		07: GEO.IP4 := IP4_DECODE(STR:=CTRL.VALUE); (* IP-Adresse *)
		10: GEO.STATE := 'OK' = CTRL.VALUE; (* STATUS *)
		13: GEO.COUNTRY_CODE := CTRL.VALUE; (* Country-Code *)
		16: GEO.COUNTRY_NAME := CTRL.VALUE; (* Country-Name *)
		19: GEO.REGION_CODE := CTRL.VALUE; (* Region-Code *)
		22: GEO.REGION_NAME := CTRL.VALUE; (* Region-Name *)
		25: GEO.CITY := CTRL.VALUE; (* City *)
		31: GEO.GEO_LATITUDE := value_real; (* Latitude *)
		34: GEO.GEO_LONGITUDE := value_real; (* Longitude *)
		37: GEO.TIME_ZONE_NAME := CTRL.VALUE; (* TimeZone Name *)
		40: GEO.GMT_OFFSET := value_int; (* GMT OFFSET in Sekunden *)
		43: GEO.IS_DST := value_int > 0; (* Sommerzeit aktiv *)
		END_CASE;

	ELSIF CTRL.TYP = 99 THEN (* EXIT - letztes Element gelesen *)
		DONE := TRUE;
		state := 100;
	END_IF;

100:
	(* UNLOCK HTTP DATA *)
	IF (NOT HTTP_GET.DONE) THEN
		state := 0;
		BUSY := FALSE;
		DONE := ERROR_T = BYTE#0;
	END_IF;

END_CASE;

(* ---------------- DNS --------------- *)
DNS_CLIENT(	IP_C:=IP_C,
			S_BUF:=S_BUF,
			R_BUF:=R_BUF,
			DOMAIN:=URL_DATA.DOMAIN,
			IP4_DNS:=DWORD#00,
			ACTIVATE:=state=40 (* DNS Start *)
			);

(* nicht oder nicht direkt verwendete Parameter *)
(* 	DWORD :=DNS_CLIENT.IP4;
	BOOL  :=DNS_CLIENT.DONE;
	BYTE  :=DNS_CLIENT.ERROR; *)
(* -------------------------------------*)

(* ------------- HTTP_GET --------------- *)
HTTP_GET(	IP_C:=IP_C,
			S_BUF:=S_BUF,
			R_BUF:=R_BUF,
			IP4:=DNS_CLIENT.IP4,
			GET:=state=60,
			MODE:=BYTE#2, (* HTTP 1.1 mit persistenter Verbindung *)
			UNLOCK_BUF:=state=100,
			URL_DATA:=URL_DATA
			);

(* nicht oder nicht direkt verwendete Parameter *)
(*	STRING := HTTP_GET.HTTP_STATUS;
	UINT :=HTTP_GET.HEADER_START;
	UINT :=HTTP_GET.HEADER_STOP;
	UINT :=HTTP_GET.BODY_START;
	UINT :=HTTP_GET.BODY_STOP;
	BOOL :=HTTP_GET.DONE;
	BYTE :=HTTP_GET.ERROR;
*)
(* -------------------------------------*)

last_state := ACTIVATE;

(* revision history
ks	14. aug. 2009	rev 1.0
	original version

ks	07. oct. 2010	rev 1.1
	new url , ip2geo fields , REAL_CHECK
*)

END_FUNCTION_BLOCK

// POUs/DEMO/IP2GEO_DEMO
PROGRAM IP2GEO_DEMO
VAR
	IP_C: IP_C;
	S_BUF: NETWORK_BUFFER;
	R_BUF: NETWORK_BUFFER;
	IP_CONTROL_1: IP_CONTROL;
	CLK_PRG : oscat_basic.CLK_PRG;
	IP2GEO_1: IP2GEO;
	GEO: IP2GEO_DATA;
	activate: BOOL := TRUE;
	done: BOOL;
	busy: BOOL;
	error_c: DWORD;
	error_t: BYTE;
END_VAR
VAR // added by the converter: edge detectors and wires of the graphical bodies
    _w1 : ANY;
END_VAR

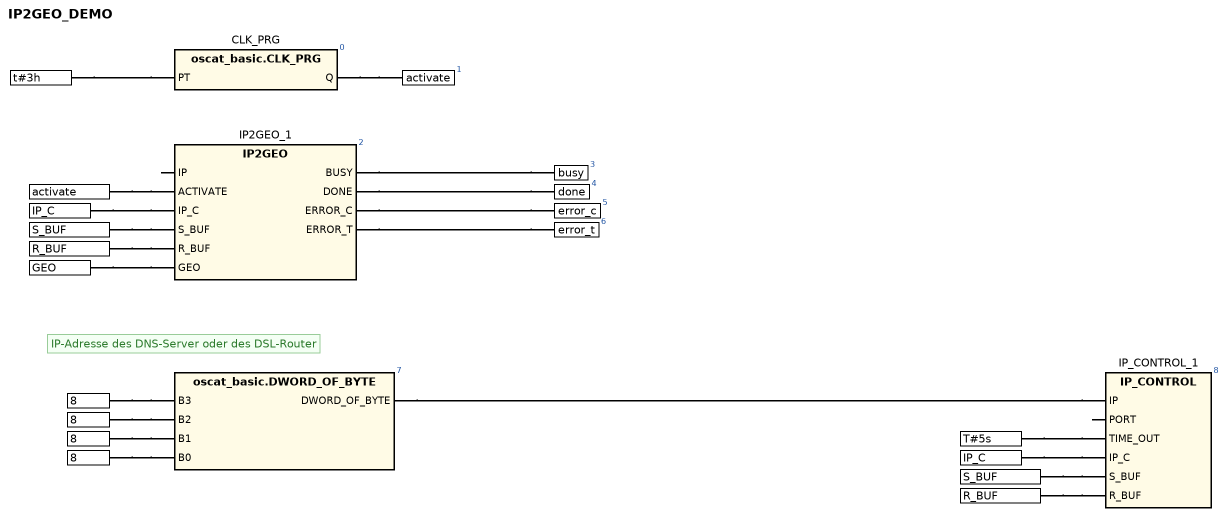
CLK_PRG(PT := t#3h); // oscat_basic.CLK_PRG
activate := CLK_PRG.Q;
IP2GEO_1(ACTIVATE := activate, IP_C := IP_C, S_BUF := S_BUF, R_BUF := R_BUF, GEO := GEO); // IP2GEO
busy := IP2GEO_1.BUSY;
done := IP2GEO_1.DONE;
error_c := IP2GEO_1.ERROR_C;
error_t := IP2GEO_1.ERROR_T;
// IP-Adresse des DNS-Server oder des DSL-Router
_w1 := oscat_basic.DWORD_OF_BYTE(B3 := 8, B2 := 8, B1 := 8, B0 := 8);
IP_CONTROL_1(IP := _w1, TIME_OUT := T#5s, IP_C := IP_C, S_BUF := S_BUF, R_BUF := R_BUF); // IP_CONTROL

END_PROGRAM

// POUs/CONVERT/IP4_CHECK
FUNCTION IP4_CHECK : BOOL
VAR_INPUT
	NIP : DWORD;
	LIP : DWORD;
	SM : DWORD;
END_VAR


(*
version 1.0	4. mar 2008
programmer 	hugo
tested by		oscat

IP4_CHECK testet ob eine Network IP und Local_IP im selben Subnet sind.

*)

IP4_CHECK := (NIP AND sm) = (LIP AND SM);


(* revision history
hm		4. mar 2008	rev 1.0
	original version

*)

END_FUNCTION

// POUs/DRIVER/IRTRANS_DECODE
FUNCTION_BLOCK IRTRANS_DECODE
VAR_IN_OUT
	IP_C : IP_C; (* IP_Control Verwaltungsstruktur *)
	R_BUF : NETWORK_BUFFER_SHORT;
END_VAR
VAR_OUTPUT
	CMD : BOOL;
	DEV : STRING;
	KEY : STRING;
	ERROR : BOOL;
END_VAR
VAR
	i : INT;
	stop : INT;
	pt : POINTER TO BYTE;
	buffer : POINTER TO ARRAY[0..32000] OF BYTE;
	size : UINT;
	z : BYTE;
END_VAR

(*

version 1.2		06. dec. 2009
programmer 		ks
tested by		ks

*)

size := R_BUF.SIZE;

(* do nothing if the buffer is empty *)
IF size > 0 AND IP_C.MAILBOX[1] <> z THEN
	i := 0;
	error := TRUE;
	stop := size - 2;
	(* read characters before first comma and store in device *)
	pt := ADR(dev);
	buffer := ADR(R_BUF.BUFFER);
	WHILE i < stop DO
		IF buffer^[i] = 44 THEN EXIT; END_IF;
		pt^ := buffer^[i];
		pt := pt + 1;
		i := i + 1;
	END_WHILE;
	(* terminate the device string *)
	pt^ := 0;
	(* read after first comma and store in key *)
	i := i + 1;
	pt := ADR(key);
	WHILE i < stop DO
		pt^ := buffer^[i];
		pt := pt + 1;
		i := i + 1;
	END_WHILE;
	(* terminate the key string *)
	pt^:= 0;
	(* check if last two characters are $R$N 13, 10 *)
	IF buffer^[i] <> 13 AND buffer^[i+1] <> 10 THEN	RETURN;	END_IF;
	(* check if device and key are present *)
	IF LEN(dev) = 0 OR LEN(key) = 0 THEN RETURN; END_IF;
	(* a valid transmission has been received *)
	cmd := TRUE;
	error := FALSE;
ELSE
	error := FALSE;
	cmd := FALSE;
END_IF;

z := IP_C.MAILBOX[1];

(* revision history
ks	18. oct. 2008	rev 1.0
	original version
ks	20. oct. 2009	rev 1.1
	Networkbuffer und Buffer-funktionen auf Basis 0
ks	06. dec. 2009	rev 1.2
	Codeanpassung für IRTRANS_SERVER
*)

END_FUNCTION_BLOCK

// POUs/DRIVER/IRTRANS_SERVER
FUNCTION_BLOCK IRTRANS_SERVER
VAR_IN_OUT
	IP_C : IP_C; (* IP_Control Verwaltungsstruktur *)
	S_BUF : NETWORK_BUFFER_SHORT;
	R_BUF : NETWORK_BUFFER_SHORT;
END_VAR
VAR_INPUT
	UDP_TCP : BOOL;
END_VAR
VAR_OUTPUT
	S_ENABLE : BOOL;
	R_ENABLE : BOOL;
	ERROR : DWORD;
END_VAR
VAR
	t : TON;
END_VAR

(*
version 1.1		17. may. 2011
programmer 		ks
tested by			ks
*)

IF NOT IP_C.C_ENABLE THEN
	(* IP Datenverkehr einrichten *)
	IP_C.C_PORT := WORD#0; (* Portnummer eintragen *)
	IP_C.C_IP := DWORD#00; (* IP eintragen *)
	IP_C.C_MODE := SEL(UDP_TCP,5,4); (* 4 = Mode: TCP+PASSIV+PORT / 5 = Mode: UDP+PASSIV+PORT*)
	IP_C.C_ENABLE := TRUE; (* Verbindungsaufbau freigeben *)
	IP_C.R_OBSERVE := FALSE; (* Datenempfang ueberwachen *)
	IP_C.TIME_RESET := TRUE; (* Zeitueberwachung rücksetzen *)
	S_BUF.SIZE := UINT#0; (* Sendedaten rücksetzen *)
	R_BUF.SIZE := UINT#0; (* Empfangsdaten rücksetzen *)
END_IF;

R_ENABLE := IP_C.C_STATE > 127;
S_ENABLE := R_ENABLE AND (IP_C.MAILBOX[1] > 0 OR IP_C.C_MODE <> 5);
ERROR := IP_C.ERROR;

t(IN:= IP_C.ERROR > 0, PT:=T#5s);
IF t.Q THEN
	IP_C.TIME_RESET := TRUE; (* Error Reset *)
END_IF;

(* revision history
ks	6. dec 2009		rev 1.0
	original version

ks	17. may 2011		rev 1.1
	neue Fehlerausgabe und Empfangsbuffer rücksetzen
*)

END_FUNCTION_BLOCK

// POUs/DEMO/IRTRANS_DEMO
PROGRAM IRTRANS_DEMO
VAR
	IP_C : IP_C;
	S_BUF : NETWORK_BUFFER_SHORT;
	R_BUF : NETWORK_BUFFER_SHORT;
	IP_CONTROL2 : IP_CONTROL2;
	IRTRANS_DECODE : IRTRANS_DECODE;
	IRTRANS_RCV_4 : IRTRANS_RCV_4;
	DRIVER_4 : oscat_basic.DRIVER_4;
	IRTRANS_SERVER : IRTRANS_SERVER;
	IRTRANS_SND_8_1 : IRTRANS_SND_8;
	IRTRANS_SND_8_2 : IRTRANS_SND_8;
	Q0: BOOL;
	Q1: BOOL;
	Q2: BOOL;
	Q3: BOOL;
	error: BOOL;
	error_server: DWORD;
	Send_1_0: BOOL := TRUE;
	Send_1_1: BOOL;
	Send_1_2: BOOL;
	Send_1_3: BOOL;
	Send_1_4: BOOL;
	Send_1_5: BOOL;
	Send_1_6: BOOL;
	Send_1_7: BOOL;
	Send_2_0: BOOL := TRUE;
	Send_2_1: BOOL;
	Send_2_2: BOOL;
	Send_2_3: BOOL;
	Send_2_4: BOOL;
	Send_2_5: BOOL;
	Send_2_6: BOOL;
	Send_2_7: BOOL;
	R_ENABLE: BOOL;
	S_ENABLE: BOOL;
	MODE: BOOL := FALSE;
	KEY_1: BYTE;
	KEY_2: BYTE;
END_VAR

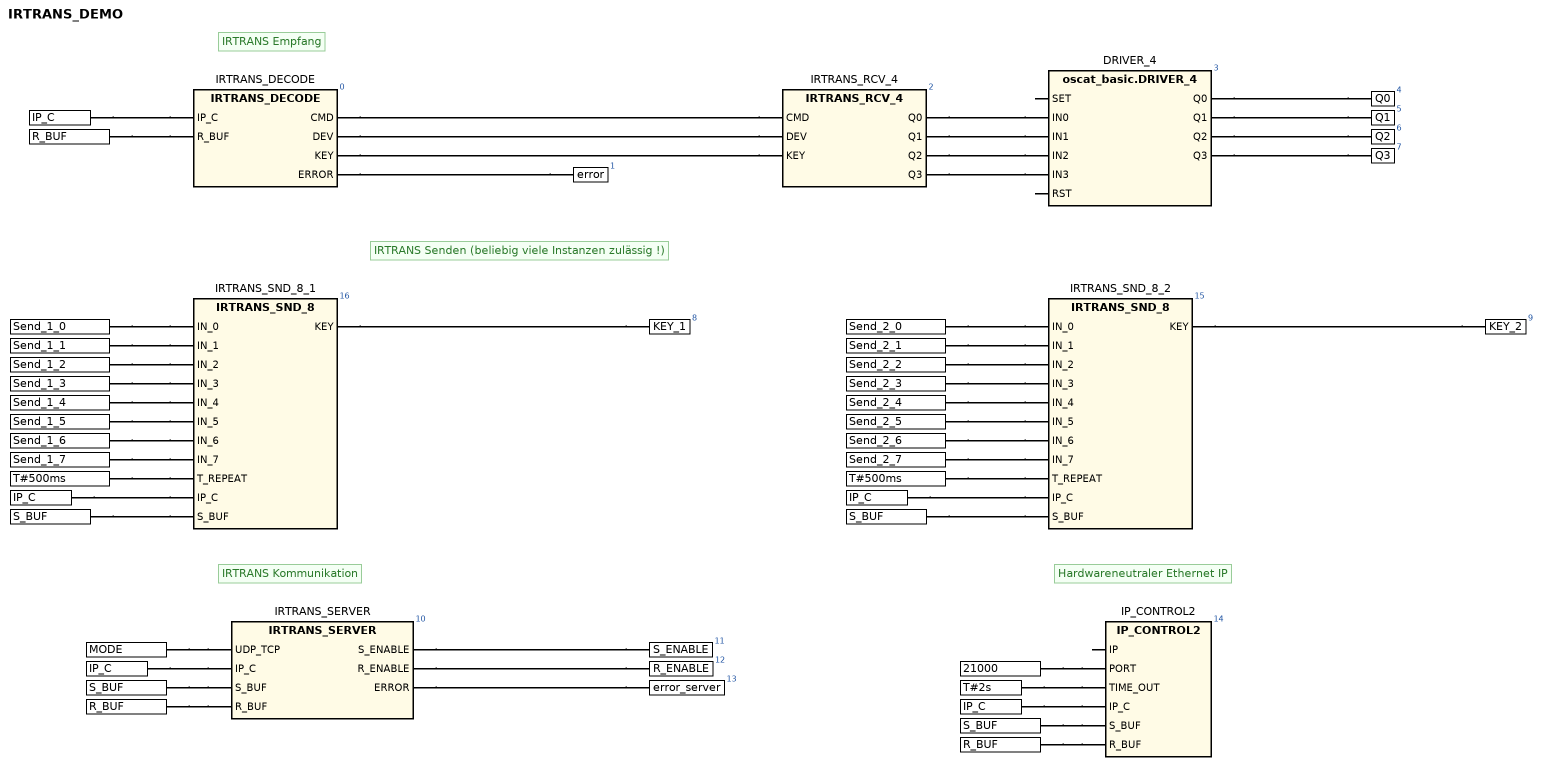
// note: 21 stored wires end on pins the file does not list and are not shown
// IRTRANS Empfang
IRTRANS_DECODE(IP_C := IP_C, R_BUF := R_BUF);
error := IRTRANS_DECODE.ERROR;
IRTRANS_RCV_4(CMD := IRTRANS_DECODE.CMD, DEV := IRTRANS_DECODE.DEV, KEY := IRTRANS_DECODE.KEY);
DRIVER_4(IN0 := IRTRANS_RCV_4.Q0, IN1 := IRTRANS_RCV_4.Q1, IN2 := IRTRANS_RCV_4.Q2, IN3 := IRTRANS_RCV_4.Q3); // oscat_basic.DRIVER_4
Q0 := DRIVER_4.Q0;
Q1 := DRIVER_4.Q1;
Q2 := DRIVER_4.Q2;
Q3 := DRIVER_4.Q3;
KEY_1 := IRTRANS_SND_8_1.KEY;
KEY_2 := IRTRANS_SND_8_2.KEY;
// IRTRANS Kommunikation
IRTRANS_SERVER(UDP_TCP := MODE, IP_C := IP_C, S_BUF := S_BUF, R_BUF := R_BUF);
S_ENABLE := IRTRANS_SERVER.S_ENABLE;
R_ENABLE := IRTRANS_SERVER.R_ENABLE;
error_server := IRTRANS_SERVER.ERROR;
// Hardwareneutraler Ethernet IP
IP_CONTROL2(PORT := 21000, TIME_OUT := T#2s, IP_C := IP_C, S_BUF := S_BUF, R_BUF := R_BUF);
IRTRANS_SND_8_2(
    IN_0 := Send_2_0,
    IN_1 := Send_2_1,
    IN_2 := Send_2_2,
    IN_3 := Send_2_3,
    IN_4 := Send_2_4,
    IN_5 := Send_2_5,
    IN_6 := Send_2_6,
    IN_7 := Send_2_7,
    T_REPEAT := T#500ms,
    IP_C := IP_C,
    S_BUF := S_BUF); // IRTRANS_SND_8
// IRTRANS Senden (beliebig viele Instanzen zulässig !)
IRTRANS_SND_8_1(
    IN_0 := Send_1_0,
    IN_1 := Send_1_1,
    IN_2 := Send_1_2,
    IN_3 := Send_1_3,
    IN_4 := Send_1_4,
    IN_5 := Send_1_5,
    IN_6 := Send_1_6,
    IN_7 := Send_1_7,
    T_REPEAT := T#500ms,
    IP_C := IP_C,
    S_BUF := S_BUF); // IRTRANS_SND_8

END_PROGRAM

// POUs/DRIVER/IRTRANS_RCV_4
FUNCTION_BLOCK IRTRANS_RCV_4
VAR_INPUT CONSTANT
	DEV_CODE : STRING;
	KEY_CODE_0 : STRING;
	KEY_CODE_1 : STRING;
	KEY_CODE_2 : STRING;
	KEY_CODE_3 : STRING;
END_VAR
VAR_INPUT
	CMD : BOOL;
END_VAR
VAR_IN_OUT
	DEV : STRING;
	KEY : STRING;
END_VAR
VAR_OUTPUT
	Q0, Q1, Q2, Q3 : BOOL;
END_VAR
VAR_TEMP
	decode: BOOL;
END_VAR

(*

version 1.3	06. dec. 2009
programmer 	hugo
tested BY	oscat

*)

decode := cmd AND dev_code = dev;

Q0 := key = key_code_0 AND decode;
Q1 := key = key_code_1 AND decode;
Q2 := key = key_code_2 AND decode;
Q3 := key = key_code_3 AND decode;



(* revision history
hm	2. jan 2008		rev 1.0
	original version

hm	17. oct. 2008	rev 1.1
	improved performance

hm	19. oct. 2008	rev 1.2
	changed input device_code to dev_code and device to dev for compatibility reasons

hm	06. dec. 2008	rev 1.3
	IRTRANS_1 renamed to IRTRANS_RCV_4

*)

END_FUNCTION_BLOCK

// POUs/HARDWARE/IP_CONTROL2
FUNCTION_BLOCK IP_CONTROL2
VAR_IN_OUT
	IP_C : IP_C; (* IP_Control Verwaltungsstruktur *)
	S_BUF : NETWORK_BUFFER_SHORT; (* Externer Sendbuffer *)
	R_BUF : NETWORK_BUFFER_SHORT; (* Externer Receivebuffer *)
END_VAR
VAR_INPUT
	IP : DWORD; (* IP Adresse *)
	PORT : WORD; (* Port Nummer *)
	TIME_OUT : TIME; (* Ueberwachungszeit Connect / Send / Receive *)
END_VAR
VAR
	c_time : UDINT; (* CONNECT-Time (Zeit bei nicht vorhandener Verbindung) *)
	s_time : UDINT; (* SEND-Time    (Zeit seit letzten Datensenden) *)
	r_time : UDINT; (* RECEIVE-Time (Zeit seit letztem Datenempfang) *)

	c_enable : BOOL; (* Connect: freigabe *)
	c_ip : DWORD; (* Connect: aktuelle IP-Adresse *)
	c_port : WORD; (* Connect: aktuelle Port-Nummer *)
	c_mode : BYTE; (* Connect: aktueller Mode UDP/TCP...... *)
	c_status : BYTE; (* Connect: Status (Errorcode) *)
	c_ready : BOOL; (* Connect: Verbindung aufgebaut *)
	c_ready_old : BOOL; (* Connect: letzter Zustand von c_ready für Flankenauswertung *)
	c_select : BOOL; (* non blocking mode - abfrage über select durchführen *)
	c_fdWrite : SOCKET_FD_SET;
	c_Timeout : SOCKET_TIMEVAL;

	s_total : INT; (* Send: Gesamtanzahl Bytes zum senden *)
	s_cur_pos : INT; (* Send: aktuelle Sendeposition *)
	s_cur_size : INT; (* Send: aktuelle Sendegroesse *)
	s_max_size : INT; (* Send: maximale Telegrammlänge fuer Senden *)
	s_start : BOOL; (* Send: Sende modus aktivieren *)
	s_active : BOOL; (* Send: Daten senden ist aktiv *)
	s_req : BOOL; (* Send: Start Daten senden *)
	s_done : BOOL; (* Send: ohne Fehler beendet *)
	s_status : BYTE; (* Send: Status (Errorcodes) *)

	r_status : BYTE; (* Receive: Status (Errorcodes) *)
	r_count : INT; (* Receive: Anzahl empfangener Bytes *)
	r_offset : INT; (* Receive: aktuelle Position in externen Receivebuffer *)
	r_max_size : INT; (* Receive: groesse des externen Empfangbuffers*)

	new_connection : BOOL; (* Neue Verbindungsparameter vorhanden *)
	tx : DWORD; (* letzter zeitwert *)
	error_time : DWORD; (* aktueller Timeout-Wert *)

	state: BYTE; (* schrittmerker für connect *)
	server_socket : DINT:= SOCKET_INVALID;
	socket : DINT:= SOCKET_INVALID;
	sockaddr : SOCKADDRESS;
	sockaddr_size : DWORD;
	plc_841 : BOOL;
	plc_881 : BOOL;
	dint_true : DINT := 1;
	bytes_received : DINT;
	bytes_sent : DINT;
	udp_mode : BOOL;

	(*LOG_MSG : LOG_MSG;
	_debug_enable : BOOL := TRUE;
	debug_index : INT;
	debug_ID : INT;
	debug_lasterror : DWORD;
	debug_last_id : INT := 255;
	state_last: BYTE;*)

END_VAR

VAR CONSTANT
	STOP : BYTE := 0;
	TS_INIT: BYTE := 1;
	TS_OPEN : BYTE:= 2;
	UDP_INIT : BYTE:= 31;
	TC_INIT : BYTE:= 51;
	TC_CONNECT : BYTE:= 52;
	C_WAIT : BYTE:= 250;
	C_CLOSE : BYTE:= 251;
END_VAR

(*

version 1.9		26. Feb. 2012
programmer 		ks
tested by			ks

IP_CONTROL ist ein Wrapper-Baustein um eine Hersteller neutrale Schnittstelle zum Ethernet zu schaffen
*)

(* ---------------------- Debug-Message ----------------------------*)
(*IF _debug_enable THEN
	IF IP_C.FIFO.ID > BYTE#0 THEN
		debug_index := IP_C.FIFO.NR;
		debug_ID := BYTE_TO_INT(IP_C.FIFO.X[debug_index]);
	END_IF;
END_IF;*)
(* -----------------------------------------------------------------------------*)

(* read system time *)
tx := OSCAT_BASIC.T_PLC_MS();

IF IP_C.C_PORT = 0 THEN
	IP_C.C_PORT := PORT; (* uebergebenen PORT durch parametrierten PORT ersetzen *)
END_IF;
IF IP_C.C_IP = 0 AND IP_C.C_MODE < 4 THEN
	IP_C.C_IP := IP; (* uebergebene IP durch paramtrierte IP ersetzen *)
END_IF;

new_connection := c_ip <> IP_C.C_IP OR c_mode <> IP_C.C_MODE OR c_port <> IP_C.C_PORT; (* neue Verbindungs erwünscht ? *)
c_enable := IP_C.C_ENABLE AND NOT new_connection;

IF IP_C.C_ENABLE AND IP_C.ERROR = 0 AND state = STOP THEN (* Freigabe,kein Fehler,kein Socket offen *)
	c_ip   := IP_C.C_IP;
	c_mode := IP_C.C_MODE;
	c_port := IP_C.C_PORT;
	plc_841 := SYSLIBSOCKETS_OPTION.1; (* Bit 1 = WAGO 750-841 *)
	plc_881 := SYSLIBSOCKETS_OPTION.2; (* Bit 1 = WAGO 750-881 *)
	udp_mode := C_MODE.0; (* Mode 1,3,5 = udp *)

	error_time := TIME_TO_DWORD(MAX(T#200ms,TIME_OUT));
	IP_C.TIME_RESET := TRUE; (* Alle Timer ruecksetzen *)

	r_max_size := SIZEOF(R_BUF.BUFFER);
	s_max_size := SIZEOF(S_BUF.BUFFER);

	IF C_MODE.0 THEN (* Mode: 1,3,5 = UDP CLIENT/SERVER *)
		state := UDP_INIT;
	ELSIF C_MODE = 0 THEN (* Mode: 0 = TCP CLIENT *)
		state := TC_INIT;
	ELSE
		state := TS_INIT; (* Mode: 2,4 = TCP SERVER *)
	END_IF;

	(* ---------------------- Debug-Message ----------------------------*)
	(*IF _debug_enable THEN
		LOG_CL.NEW_MSG := 'IP_CON: MODE ~1 / IP ~2 / PORT ~3 /ID ~6';
		LOG_CL.PRINTF[1] := BYTE_TO_STRING(C_MODE);
		LOG_CL.PRINTF[2] := IP4_TO_STRING(c_ip);
		LOG_CL.PRINTF[3] := WORD_TO_STRING(c_port);
		LOG_CL.PRINTF[6] := INT_TO_STRING(debug_ID);
		LOG_MSG();
	END_IF;*)
	(* -----------------------------------------------------------------------------*)

END_IF;

(* ---------------------- Debug-Message ----------------------------*)
(*IF  _debug_enable THEN
	IF state <> state_last THEN
		LOG_CL.NEW_MSG := 'IP_STEP ~1 -IP_ID ~6';
		LOG_CL.PRINTF[1] := BYTE_TO_STRING(state);
		LOG_CL.PRINTF[6] := INT_TO_STRING(debug_ID);
		LOG_MSG();
		state_last := state;
	END_IF;
END_IF;*)
(* -----------------------------------------------------------------------------*)

IF IP_C.TIME_RESET THEN (* Alle Timer ruecksetzen *)
	IP_C.TIME_RESET := FALSE; (* Reset rücksetzen *)
	c_time := tx; (* Connect Timer ruecksetzen *)
	s_time := tx; (* Send Timer ruecksetzen *)
	r_time := tx; (* Receive Timer ruecksetzen *)

	c_status := BYTE#0; (* letzten Connect Fehler rücksetzen *)
	s_status := BYTE#0; (* letzten Send Fehler rücksetzen *)
	r_status := BYTE#0; (* letzten Receive Fehler rücksetzen *)
END_IF;

(* ---------------------------------------------- *)

CASE state OF

UDP_INIT: (* UDP_CLIENT + SERVER *)
	socket := SysSockCreate(SOCKET_AF_INET, SOCKET_DGRAM, SOCKET_IPPROTO_IP);
	IF socket < 0 THEN
		c_status := 1; (* SysSockCreate failed *)
		state := C_CLOSE;
	ELSE
		SysSockSetOption(socket, SOCKET_SOL, SOCKET_SO_BROADCAST, ADR(dint_true), SIZEOF(dint_true)); (* allow broadcast *)
		SysSockIoctl(socket, SOCKET_FIONBIO, ADR(dint_true)); (* put socket in non-blocking mode *)
		sockaddr.sin_family := SOCKET_AF_INET;
		sockaddr.sin_port := SysSockHtons(c_port);
		sockaddr.sin_addr := SEL(c_mode = 1, SOCKET_INADDR_ANY, SysSockNtohl(c_ip));

		IF c_mode >= 2 THEN (* SERVER Mode *)
			IF SysSockBind(socket, ADR(sockaddr), SIZEOF(sockaddr)) THEN
				c_ready := TRUE; (* Connected *)
				state:= C_WAIT;
			ELSE
				c_status := 2; (* SysSockBind failed *)
				state := C_CLOSE;
			END_IF;
		ELSE
			c_ready := TRUE; (* Connected *)
			state:= C_WAIT;
		END_IF;
	END_IF;

(* ---------------------------------------------- *)

TC_INIT: (* TCP-CLIENT (AKTIV) *)
	socket := SysSockCreate(SOCKET_AF_INET, SOCKET_STREAM, SOCKET_IPPROTO_IP);
	IF socket < 0 THEN
		c_status := 1;  (* SysSockCreate failed *)
		state := C_CLOSE;
	ELSE
		IF plc_841 OR plc_881 THEN
			SysSockSetOption(socket,6,SOCKET_TCP_NODELAY, ADR(dint_true), SIZEOF(dint_true)); (* Set Push-Bit *)
		END_IF;
		SysSockIoctl(socket, SOCKET_FIONBIO, ADR(dint_true)); (* NonBlocking mode *)
		sockaddr.sin_family := SOCKET_AF_INET;
		sockaddr.sin_port := SysSockNtohs(c_port);
		sockaddr.sin_addr := SysSockNtohl(c_ip);
		c_select := FALSE;
		state := TC_CONNECT;
	END_IF;

(* ---------------------------------------------- *)

TC_CONNECT:
	IF NOT c_enable OR c_status = 255 THEN (* keine freigabe oder connect timeout *)
			state:= C_CLOSE;
	ELSE
		IF c_select = FALSE THEN
			IF SysSockConnect(socket,ADR(sockaddr),SIZEOF(sockaddr)) THEN
				c_ready := TRUE; (* Connected *)
				state:= C_WAIT;
			ELSE
				(* Connect durchgeführt, aber noch nicht verbunden, dann optional mit select-abfrage weitermachen *)
				c_select := SYSLIBSOCKETS_OPTION.0; (* Bit 0 = TCP-Client - use SysSockselect *)
			END_IF;
		ELSE
			c_Timeout.tv_sec := 0;
			c_Timeout.tv_usec := 0;
			c_fdWrite.fd_count := 1;
			c_fdWrite.fd_array[0] := socket;
			IF SysSockSelect(SOCKET_FD_SETSIZE,0,ADR(c_fdWrite),0, ADR(c_Timeout)) > 0 THEN
				c_ready := TRUE; (* Connected *)
				state:= C_WAIT;
			END_IF;
		END_IF;
	END_IF;

(* ---------------------------------------------- *)

TS_INIT: (* TCP-SERVER (PASSIV) *)
	server_socket := SysSockCreate(SOCKET_AF_INET, SOCKET_STREAM, SOCKET_IPPROTO_IP); (* Create Socket *)
	IF server_socket = SOCKET_INVALID THEN
		c_status := 1; (* SysSockCreate failed *)
		state:= C_CLOSE;
	ELSE (* Address bindings *)
		SysSockSetOption( server_socket, SOCKET_SOL, SOCKET_SO_REUSEADDR, ADR(dint_true), SIZEOF(dint_true) );
		sockaddr.sin_family:= SOCKET_AF_INET;
		sockaddr.sin_port := SysSockHtons(c_port);
		sockaddr.sin_addr := SOCKET_INADDR_ANY;
		IF NOT SysSockBind(server_socket, ADR(sockaddr), SIZEOF(sockaddr)) THEN
			c_status := 2; (* SysSockBind failed *)
			state := C_CLOSE;
		ELSIF NOT SysSockListen(server_socket, 1) THEN (* erzeugt Warteschlange für eine Verbindung *)
			c_status := 3; (* SysSockListen failed *)
			state:= C_CLOSE;
		ELSE
			SysSockIoctl(server_socket, SOCKET_FIONBIO, ADR(dint_true)); (* NonBlocking mode *)
			state:= TS_OPEN;
		END_IF;
	END_IF;

(* ---------------------------------------------- *)

TS_OPEN: (* Waiting for incomming connection *)
	sockaddr_size := SIZEOF(sockaddr);
	socket := SysSockAccept(server_socket, ADR(sockaddr), ADR(sockaddr_size));

	IF socket <> SOCKET_INVALID THEN (* neuer Verbindungswunsch vorhanden *)
		IF c_mode = BYTE#2 AND sockaddr.sin_addr <> SysSockNtohl(c_ip) THEN (* Mode 2 = TCP + PASSIVE + PORT + IP  auf richtige Partner-IP prüfen *)
			state:= C_CLOSE;
		ELSE
			IF plc_841 OR plc_881 THEN
				SysSockSetOption(socket, 6, SOCKET_TCP_NODELAY, ADR(dint_true), SIZEOF(dint_true)); (* Set Push-Bit *)
			END_IF;
			SysSockIoctl(socket, SOCKET_FIONBIO, ADR(dint_true)); (* NonBlocking mode *)
			c_ready := TRUE; (* Connected *)
			state := C_WAIT;
		END_IF;
	ELSIF NOT c_enable THEN (* keine freigabe mehr ? *)
			state:= C_CLOSE;
	END_IF;

(* ---------------------------------------------- *)

C_WAIT: (* Warten auf Anforderung für Beenden *)
	IF NOT c_enable OR NOT c_ready THEN
		state:= C_CLOSE;
	END_IF

(* ---------------------------------------------- *)

C_CLOSE: (* Close the Sockets *)
	c_ready := FALSE;
	IF socket >= 0 THEN
		IF (NOT plc_841) AND (NOT plc_881) THEN
			SysSockShutdown(socket, 0); (* 870 *)
		END_IF;
		SysSockClose(socket);
		socket := SOCKET_INVALID;
	END_IF
	IF server_socket >= 0 THEN
		IF (NOT plc_841) AND (NOT plc_881) THEN
			SysSockShutdown(server_socket, 0); (* 870 *)
		END_IF;
		SysSockClose(server_socket);
		server_socket := SOCKET_INVALID;
	END_IF
	state:= STOP;
END_CASE;

(* ---------------------------------------------- *)

IF c_ready THEN
	IF NOT c_ready_old THEN (* Verbindung aufgebaut - positive Flanke erkannt *)
		IP_C.C_STATE := 254;
		IP_C.TIME_RESET := TRUE; (* Alle Timer ruecksetzen *)
		(* ---------------------- Debug-Message ----------------------------*)
		(*IF _debug_enable THEN
			LOG_CL.NEW_MSG := 'IP_CON: CONNECTED -IP_ID ~6';
			LOG_CL.PRINTF[6] := INT_TO_STRING(debug_ID);
			LOG_MSG();
		END_IF;*)
		(* -----------------------------------------------------------------------------*)
	ELSE
		IP_C.C_STATE := 255; (* Verbindung ist aufgebaut *)
	END_IF;
ELSE
	IF c_ready_old THEN (* Verbindung abgebaut - negative Flanke erkannt *)
		IP_C.C_STATE := 1;
		IP_C.MAILBOX[1] := 0; (* Receive Info rücksetzen *)
		IP_C.MAILBOX[2] := 0; (* Send-Pause rücksetzen *)
		IP_C.MAILBOX[3] := 0; (* Receive-Pause rücksetzen *)
		IF NOT new_connection THEN
			s_active := FALSE; (* Sendeaktivitäten stoppen *)
			s_req := FALSE; (* Sendefreigabe rücksetzen *)
			S_BUF.SIZE := 0; (* Sendelänge löschen *)
			(* IP_C.TIME_RESET := TRUE; *) (* Alle Timer ruecksetzen *)
		END_IF;
		(* ---------------------- Debug-Message ----------------------------*)
		(*IF _debug_enable THEN
			LOG_CL.NEW_MSG := 'IP_CON: DISCONNECTED';
			LOG_MSG();
		END_IF;*)
		(* -----------------------------------------------------------------------------*)
	ELSE
		IP_C.C_STATE := 0; (* Verbindung ist abgebaut *)
	END_IF;
END_IF;

c_ready_old := c_ready;

(* Der Datenempfang wird angehalten solange ein Sendevorgang läuft *)
(* sonst kann es vorkommen das die Antwort-daten schon empfangen werden, *)
(* bevor der Sendevorgang vom programm abgeschlossen wurde *)

IF c_ready AND NOT s_active AND IP_C.MAILBOX[3] = 0 THEN
	IF R_BUF.SIZE >= INT_TO_UINT(r_max_size) THEN
		R_BUF.SIZE := UINT#0;
		r_status := 254; (* Empfangsbuffer wegen Überlauf rückgesetzt *)
	END_IF;

	r_offset := SEL(udp_mode,UINT_TO_INT(R_BUF.SIZE),0);
	r_count := r_max_size - r_offset;

	IF udp_mode THEN
		bytes_received := SysSockRecvFrom(socket, ADR(R_BUF.BUFFER), r_count, 0, ADR(sockaddr), SIZEOF(sockaddr));

		IF c_mode = BYTE#3 AND sockaddr.sin_addr <> SysSockNtohl(c_ip) THEN (* Mode 3 = UDP + PASSIVE + PORT + IP  auf richtige Partner-IP prüfen *)
			bytes_received := 0;
			R_BUF.SIZE := UINT#0;
			sockaddr.sin_port := SysSockNtohs(c_port);
			sockaddr.sin_addr := SysSockNtohl(c_ip);
		END_IF;

	ELSE
		bytes_received := SysSockRecv(socket, ADR(R_BUF.BUFFER[r_offset]), r_count, 0);
	END_IF;

	(*UDP: IPC returns -1 if no data available or error occured,841 returns -1 if error occured and 0 if no data available*)
	CASE bytes_received OF
	-2147483648..-1: ; (* No data available or error occured *)
	 0: IF NOT udp_mode THEN (* TCP-Mode: socket wurde von remote geschlossen *)
			c_status := 253;
			c_ready := FALSE;
		END_IF;
	ELSE (* daten wurden empfangen *)
  		r_time := tx; (* Receive Timer ruecksetzen *)
		R_BUF.SIZE := INT_TO_UINT(r_offset + DINT_TO_UINT(bytes_received)); (* aktuelle buffersize eintragen *)
		IP_C.MAILBOX[1] := IP_C.MAILBOX[1] + 1; (* Receive Info *)
		IF IP_C.MAILBOX[1] = 0 THEN IP_C.MAILBOX[1] := 1; END_IF;

		(* ---------------------- Debug-Message ----------------------------*)
		(*IF _debug_enable THEN
			LOG_CL.NEW_MSG := 'IP_REC DATA: POS: ~1 : SIZE: ~2 TOTAL ~3 -IP_ID ~6';
			LOG_CL.PRINTF[1] := INT_TO_STRING(r_offset);
			LOG_CL.PRINTF[2] := INT_TO_STRING(r_count);
			LOG_CL.PRINTF[3] := UINT_TO_STRING(R_BUF.SIZE);
			LOG_CL.PRINTF[6] := INT_TO_STRING(debug_ID);
			LOG_MSG();
		END_IF;*)
		(* -----------------------------------------------------------------------------*)

	END_CASE
END_IF;

(* ---------------------------------------------- *)

IF S_BUF.SIZE > 0 THEN
	IF c_ready AND c_enable THEN
		IF NOT s_active AND IP_C.MAILBOX[2] = 0 THEN
			(* Gesamtanzahl an Bytes limitieren und uebergeben *)
			s_total := LIMIT(0,UINT_TO_INT(S_BUF.SIZE),r_max_size);
			s_cur_pos  := 0;
			s_cur_size := 0;
			s_start := TRUE; (* Daten kopieren und senden anstossen *)
			s_active := TRUE; (* Sende-Betrieb aktivieren *)
			(* ---------------------- Debug-Message ----------------------------*)
			(*IF _debug_enable THEN
				LOG_CL.NEW_MSG := 'IP_SEN INIT: TOTAL: ~1 -IP_ID ~6';
				LOG_CL.PRINTF[1] := INT_TO_STRING(S_TOTAL);
				LOG_CL.PRINTF[6] := INT_TO_STRING(debug_ID);
				LOG_MSG();
			END_IF;*)
			(* -----------------------------------------------------------------------------*)
		END_IF;

		IF s_done OR s_start THEN (* Daten senden aktiv *)

			s_start := FALSE;
			s_cur_pos := s_cur_pos + s_cur_size; (* neue Sende-Datenposition bestimmen *)
			IF s_total > s_cur_pos THEN (* weitere Daten zum senden vorhanden ? *)
				s_cur_size := s_total - s_cur_pos;
				s_cur_size := LIMIT(0, s_cur_size, s_max_size); (* Telegrammlänge begrenzen *)

				(* ---------------------- Debug-Message ----------------------------*)
				(*IF _debug_enable THEN
					LOG_CL.NEW_MSG := 'IP_SEN DATA: POS: ~1 : SIZE: ~2 TOTAL ~3 -IP_ID ~6';
					LOG_CL.PRINTF[1] := INT_TO_STRING(S_CUR_POS);
					LOG_CL.PRINTF[2] := INT_TO_STRING(S_CUR_SIZE);
					LOG_CL.PRINTF[3] := INT_TO_STRING(S_TOTAL);
					LOG_CL.PRINTF[6] := INT_TO_STRING(debug_ID);
					LOG_MSG();
				END_IF;*)
				(* -----------------------------------------------------------------------------*)

				s_time := tx; (* Send Timer ruecksetzen *)
				r_time := tx; (* Receive Timer ruecksetzen *)
				s_req := TRUE;

			ELSE
				(* keine weitere Sendedaten vorhanden -> Senden beenden *)
				s_req := FALSE;
				s_active := FALSE;
				S_BUF.SIZE := 0;
				(* ---------------------- Debug-Message ----------------------------*)
				(*IF _debug_enable THEN
					LOG_CL.NEW_MSG := 'IP_SEN FINISH -IP_ID ~6';
					LOG_CL.PRINTF[6] := INT_TO_STRING(debug_ID);
					LOG_MSG();
				END_IF;*)
				(* -----------------------------------------------------------------------------*)
			END_IF;
		END_IF;
	END_IF;
END_IF;

IF s_req THEN
	s_done := FALSE;
	IF udp_mode THEN
		bytes_sent := SysSockSendTo(socket, ADR(S_BUF.BUFFER[s_cur_pos]), s_cur_size, 0, ADR(sockaddr), SIZEOF(sockaddr));
	ELSE
		bytes_sent := SysSockSend(socket, ADR(S_BUF.BUFFER[s_cur_pos]), s_cur_size, 0);
	END_IF;

	CASE bytes_sent OF
	-2147483648..-1:	; (* ERROR: Noch nicht bereit um Daten aufzunehmen -> nächsten Zyklus wieder probieren *)
	 0: IF NOT udp_mode THEN (* TCP-Mode: socket wurde von remote geschlossen *)
			c_status := 253;
			c_ready := FALSE;
		END_IF;
	ELSE
		s_done := TRUE;
		s_cur_size := DINT_TO_INT(bytes_sent); (* Anzahl der wirklich versendeten Bytes übernehmen *)
		(* ---------------------- Debug-Message ----------------------------*)
		(*IF _debug_enable THEN
			LOG_CL.NEW_MSG := 'IP_SEN SEND_COUNT ~1 -IP_ID ~6';
			LOG_CL.PRINTF[1] := DINT_TO_STRING(s_cur_size);
			LOG_CL.PRINTF[6] := INT_TO_STRING(debug_ID);
			LOG_MSG();
		END_IF;*)
		(* -----------------------------------------------------------------------------*)
	END_CASE
END_IF;

(* ---------------------------------------------- *)

IF IP_C.R_OBSERVE = FALSE OR s_active THEN
    r_time := tx;
END_IF;

IF c_status = 0 AND tx - c_time > error_time AND c_enable AND NOT c_ready AND c_mode < 2 THEN (* Connect Timeout *)
	c_status := 255; (* Timeout-Fehler ausgeben *)
END_IF;
IF s_status = 0 AND tx - s_time > error_time AND s_active THEN (* Send Timeout *)
	s_status := 255; (* Timeout-Fehler ausgeben *)
END_IF;
IF r_status = 0 AND tx - r_time > error_time AND c_ready AND IP_C.R_OBSERVE THEN (* Receive Timeout *)
	r_status := 255; (* Timeout-Fehler ausgeben *)
END_IF;

IP_C.ERROR := OSCAT_BASIC.DWORD_OF_BYTE(c_status,s_status,r_status,0);

(* ---------------------- Debug-Message ----------------------------*)
(*IF  _debug_enable THEN
	IF (IP_C.ERROR <> debug_lasterror) THEN
		LOG_CL.NEW_MSG := 'IP_ERROR ~1 -IP_ID ~6';
		LOG_CL.PRINTF[1] := DWORD_TO_STRING(IP_C.ERROR);
		LOG_CL.PRINTF[6] := INT_TO_STRING(debug_ID);
		LOG_MSG();

		debug_lasterror := IP_C.ERROR;
		debug_last_id := debug_ID;
	END_IF;
END_IF;*)
(* -----------------------------------------------------------------------------*)

(* revision history
ks	18. oct. 2008	rev 1.0
	original version
ks	05. jan. 2009	rev 1.1
	zusätzlichen Parameter "Port" hinzugefügt, und Code bei Verbindungsaufbau angepasst
ks	28. feb. 2009	rev 1.2
	connect code angepasst und verkürzung der zyklen bei Send
ks	20. oct. 2009	rev 1.3
	network_buffer basis 0
ks	06. dec. 2009	rev 1.4
	receive_count MAILBOX[1]
ks	10. nov. 2010	rev 1.5
	send_pause MAILBOX[2] and receive_pause MAILBOX[3] 
ks	07. feb. 2011	rev 1.6
	Fehlercode 253 bei Remote-Verbindungsabbruch 
ks	30. may. 2011	rev 1.7
	Fehler bei Empfangsüberwachung
ks	26. july. 2011	rev 1.8
	Error-Reset, diverse optimierungen 
ks	26. feb. 2012	rev 1.9
	Code-Optimierung für höhere kompatibilität
*)

END_FUNCTION_BLOCK

// POUs/DRIVER/IRTRANS_SND_8
FUNCTION_BLOCK IRTRANS_SND_8
VAR_INPUT CONSTANT
	DEV_CODE : STRING;
	KEY_CODE_0 : STRING;
	KEY_CODE_1 : STRING;
	KEY_CODE_2 : STRING;
	KEY_CODE_3 : STRING;
	KEY_CODE_4 : STRING;
	KEY_CODE_5 : STRING;
	KEY_CODE_6 : STRING;
	KEY_CODE_7 : STRING;
END_VAR
VAR_INPUT
	IN_0 : BOOL;
	IN_1 : BOOL;
	IN_2 : BOOL;
	IN_3 : BOOL;
	IN_4 : BOOL;
	IN_5 : BOOL;
	IN_6 : BOOL;
	IN_7 : BOOL;
	T_REPEAT : TIME;
END_VAR
VAR_IN_OUT
	IP_C : IP_C; (* IP_Control Verwaltungsstruktur *)
	S_BUF : NETWORK_BUFFER_SHORT;
END_VAR
VAR_OUTPUT
	KEY : BYTE;
END_VAR
VAR
	skey : STRING;
	size : INT;
	str : STRING;
	t : TON;
	k : BYTE;
	lk : BYTE;
	d : BOOL;
END_VAR

(*
version 1.0		06. dec. 2009
programmer 		ks
tested by		ks
*)

d := IP_C.C_STATE > 127 AND (IP_C.MAILBOX[1] > 0 OR IP_C.C_MODE <> 5);
IF NOT d THEN RETURN; END_IF;

t(IN:= lk = k , PT:=T_REPEAT);

IF S_BUF.SIZE = 0 THEN
	IF IN_0 THEN
		skey := KEY_CODE_0; k := 1;
	ELSIF IN_1 THEN
		skey := KEY_CODE_1; k := 2;
	ELSIF IN_2 THEN
		skey := KEY_CODE_2; k := 3;
	ELSIF IN_3 THEN
		skey := KEY_CODE_3; k := 4;
	ELSIF IN_4 THEN
		skey := KEY_CODE_4; k := 5;
	ELSIF IN_5 THEN
		skey := KEY_CODE_5; k := 6;
	ELSIF IN_6 THEN
		skey := KEY_CODE_6; k := 7;
	ELSIF IN_7 THEN
		skey := KEY_CODE_7; k := 8;
	ELSE
		lk := 0;
		KEY := 0;
		RETURN; (* beenden wenn kein Key aktiv *)
	END_IF;

	IF lk <> k OR T.Q THEN (* anderer Key oder repeat wartezeit abgelaufen *)
		str := CONCAT('snd ',dev_code);
		str := CONCAT(str,',');
		str := CONCAT(str,skey);
		size := LEN(str);
		OSCAT_BASIC._STRING_TO_BUFFER(STR:=str, POS:=0, PT:=ADR(S_BUF.BUFFER), SIZE:=size);
		S_BUF.SIZE := size; (* Sendelänge eintragen *)
		KEY := k;
		lk := k; (* letzten Key speichern *)
		t(IN:=FALSE); (* Reset Time *)
	END_IF;
END_IF;

(* revision history
hm	6. dec 2009		rev 1.0
	original version
*)

END_FUNCTION_BLOCK

// POUs/DRIVER/IRTRANS_RCV_1
FUNCTION_BLOCK IRTRANS_RCV_1
VAR_INPUT CONSTANT
	DEV_CODE : STRING;
	KEY_CODE : STRING;
END_VAR
VAR_INPUT
	CMD : BOOL;
END_VAR
VAR_IN_OUT
	DEV : STRING;
	KEY : STRING;
END_VAR
VAR_OUTPUT
	Q : BOOL;
END_VAR


(*

version 1.3	06. dec. 2009
programmer 	hugo
tested by		oscat

*)

Q := cmd AND dev_code = dev AND key_code = key;

(* revision history
hm	2. jan 2008		rev 1.0
	original version

hm	20. 6. 2008		rev 1.1
	performance improvement

hm	19. oct. 2008	rev 1.2
	changed input device_code to dev_code and device to dev for compatibility reasons

hm	06. dec. 2008	rev 1.3
	IRTRANS_1 renamed to IRTRANS_RCV_1

*)

END_FUNCTION_BLOCK

// POUs/DRIVER/IRTRANS_RCV_8
FUNCTION_BLOCK IRTRANS_RCV_8
VAR_INPUT CONSTANT
	dev_code : STRING;
	key_code_0 : STRING;
	key_code_1 : STRING;
	key_code_2 : STRING;
	key_code_3 : STRING;
	key_code_4 : STRING;
	key_code_5 : STRING;
	key_code_6 : STRING;
	key_code_7 : STRING;
END_VAR
VAR_INPUT
	CMD : BOOL;
END_VAR
VAR_IN_OUT
	DEV : STRING;
	KEY : STRING;
END_VAR
VAR_OUTPUT
	Q0, Q1, Q2, Q3, Q4, Q5, Q6, Q7 : BOOL;
END_VAR
VAR_TEMP
	decode: BOOL;
END_VAR

(*

version 1.3	06. dec. 2009
programmer 	hugo
tested BY	oscat

*)

decode := cmd AND dev_code = dev;

Q0 := key = key_code_0 AND decode;
Q1 := key = key_code_1 AND decode;
Q2 := key = key_code_2 AND decode;
Q3 := key = key_code_3 AND decode;
Q4 := key = key_code_4 AND decode;
Q5 := key = key_code_5 AND decode;
Q6 := key = key_code_6 AND decode;
Q7 := key = key_code_7 AND decode;


(* revision history
hm	2. jan 2008		rev 1.0
	original version

hm	17. oct 2008	rev 1.1
	improved performance

hm	19. oct. 2008	rev 1.2
	changed input device_code to dev_code and device to dev for compatibility reasons

hm	06. dec. 2008	rev 1.3
	IRTRANS_1 renamed to IRTRANS_RCV_8

*)

END_FUNCTION_BLOCK

// POUs/DRIVER/IRTRANS_SND_1
FUNCTION_BLOCK IRTRANS_SND_1
VAR_INPUT CONSTANT
	DEV_CODE : STRING;
	KEY_CODE : STRING;
END_VAR
VAR_INPUT
	IN : BOOL;
	T_REPEAT : TIME;
END_VAR
VAR_IN_OUT
	IP_C : IP_C; (* IP_Control Verwaltungsstruktur *)
	S_BUF : NETWORK_BUFFER_SHORT;
END_VAR
VAR_OUTPUT
	KEY : BYTE;
END_VAR
VAR
	skey : STRING;
	size : INT;
	str : STRING;
	t : TON;
	k : BYTE;
	lk : BYTE;
	d : BOOL;
END_VAR

(*
version 1.0		06. dec. 2009
programmer 		ks
tested by		ks
*)

d := IP_C.C_STATE > 127 AND (IP_C.MAILBOX[1] > 0 OR IP_C.C_MODE <> 5);
IF NOT d THEN RETURN; END_IF;

t(IN:= lk = k , PT:=T_REPEAT);

IF S_BUF.SIZE = 0 THEN
	IF IN THEN
		skey := KEY_CODE; k := 1;
	ELSE
		lk := 0;
		KEY := 0;
		RETURN; (* beenden wenn kein Key aktiv *)
	END_IF;

	IF lk <> k OR T.Q THEN (* anderer Key oder repeat wartezeit abgelaufen *)
		str := CONCAT('snd ',dev_code);
		str := CONCAT(str,',');
		str := CONCAT(str,skey);
		size := LEN(str);
		OSCAT_BASIC._STRING_TO_BUFFER(STR:=str, POS:=0, PT:=ADR(S_BUF.BUFFER), SIZE:=size);
		S_BUF.SIZE := size; (* Sendelänge eintragen *)
		KEY := k;
		lk := k; (* letzten Key speichern *)
		t(IN:=FALSE); (* Reset Time *)
	END_IF;
END_IF;

(* revision history
hm	6. dec 2009		rev 1.0
	original version
*)

END_FUNCTION_BLOCK

// POUs/DRIVER/IRTRANS_SND_4
FUNCTION_BLOCK IRTRANS_SND_4
VAR_INPUT CONSTANT
	DEV_CODE : STRING;
	KEY_CODE_0 : STRING;
	KEY_CODE_1 : STRING;
	KEY_CODE_2 : STRING;
	KEY_CODE_3 : STRING;
END_VAR
VAR_INPUT
	IN_0 : BOOL;
	IN_1 : BOOL;
	IN_2 : BOOL;
	IN_3 : BOOL;
	T_REPEAT : TIME;
END_VAR
VAR_IN_OUT
	IP_C : IP_C; (* IP_Control Verwaltungsstruktur *)
	S_BUF : NETWORK_BUFFER_SHORT;
END_VAR
VAR_OUTPUT
	KEY : BYTE;
END_VAR
VAR
	skey : STRING;
	size : INT;
	str : STRING;
	t : TON;
	k : BYTE;
	lk : BYTE;
	d : BOOL;
END_VAR

(*
version 1.0		06. dec. 2009
programmer 		ks
tested by		ks
*)

d := IP_C.C_STATE > 127 AND (IP_C.MAILBOX[1] > 0 OR IP_C.C_MODE <> 5);
IF NOT d THEN RETURN; END_IF;

t(IN:= lk = k , PT:=T_REPEAT);

IF S_BUF.SIZE = 0 THEN
	IF IN_0 THEN
		skey := KEY_CODE_0; k := 1;
	ELSIF IN_1 THEN
		skey := KEY_CODE_1; k := 2;
	ELSIF IN_2 THEN
		skey := KEY_CODE_2; k := 3;
	ELSIF IN_3 THEN
		skey := KEY_CODE_3; k := 4;
	ELSE
		lk := 0;
		KEY := 0;
		RETURN; (* beenden wenn kein Key aktiv *)
	END_IF;

	IF lk <> k OR T.Q THEN (* anderer Key oder repeat wartezeit abgelaufen *)
		str := CONCAT('snd ',dev_code);
		str := CONCAT(str,',');
		str := CONCAT(str,skey);
		size := LEN(str);
		OSCAT_BASIC._STRING_TO_BUFFER(STR:=str, POS:=0, PT:=ADR(S_BUF.BUFFER), SIZE:=size);
		S_BUF.SIZE := size; (* Sendelänge eintragen *)
		KEY := k;
		lk := k; (* letzten Key speichern *)
		t(IN:=FALSE); (* Reset Time *)
	END_IF;
END_IF;

(* revision history
hm	6. dec 2009		rev 1.0
	original version
*)

END_FUNCTION_BLOCK

// POUs/CONVERT/IS_IP4
FUNCTION IS_IP4 : BOOL
VAR_INPUT
	str : STRING;
END_VAR


(*
version 1.1	10. mar 2009
programmer 	kurt
tested by		hugo

IS_IP4 testet ob ein string eine gültige IPv4 Adresse enthält.

*)

IS_IP4 := OSCAT_BASIC.COUNT_CHAR(str, 46) = 3;


(* revision history
hm	1. mar. 2008	rev 1.0
	original version

hm	10. mar. 2009	rev 1.1
	new code

*)

END_FUNCTION

// POUs/CONVERT/IS_URLCHR
FUNCTION IS_URLCHR : BOOL
VAR_INPUT
	IN : BYTE;
END_VAR


(*
version 1.0		27. apr. 2008
programmer 		hugo
tested by		hugo

IS_URL_CHR is true if a string contains only non reserved characters for an url.
the non reserved characters are : [A..Z], [a..z], [0..9], -_.~

*)

IS_URLCHR := ((IN > 47) AND (IN < 58)) OR ((IN > 64) AND (IN < 91)) OR ((IN > 96) AND (IN < 123)) OR (in = 126) OR (in = 95) OR (in =45) OR (in =46);


(* revision history
hm		27. apr. 2008	rev 1.0
	original version

*)

END_FUNCTION

// POUs/OTHER/LOG_VIEWPORT
FUNCTION_BLOCK LOG_VIEWPORT
VAR_IN_OUT
	LC : LOG_CONTROL;
	LV : us_LOG_VIEWPORT;
END_VAR
VAR
	pos : INT;
	count : INT;
	idx : INT;
	base : INT;
	update_pos : BOOL;
END_VAR

(*
version 1.1		05 mai 2012
programmer		ks
tested BY		ks

LOG_VIEWPORT erzeugt einen Liste der Meldungen des Loggingbuffers die innerhalb einer virtuellen Ansicht enthalten sind.
*)

(* Scroll Button verarbeiten *)
IF LV.MOVE_TO_X <> 0 THEN
	CASE LV.MOVE_TO_X OF
	30000: pos := 1 ; (* älteste Meldung anzeigen *)
	30001: pos := LC.SIZE; (* neueste Meldung anzeigen *)
	30002: pos := pos + LV.COUNT; (* eine Seite nach unten blättern -> Richtung neuere Nachrichten *)
	30003: pos := pos - LV.COUNT; (* eine Seite nach oben blättern -> Richtung ältere Nachrichten *)
	ELSE
		pos := pos + LV.MOVE_TO_X;
	END_CASE;
	update_pos := TRUE;
	LV.MOVE_TO_X := 0;
END_IF;

IF (LV.UPDATE_COUNT <> LC.UPDATE_COUNT) OR update_pos THEN (* Aktualisierung überwachen *)
	LV.UPDATE := TRUE;
	LV.UPDATE_COUNT := LC.UPDATE_COUNT;
	update_pos := FALSE;

	(* pos prüfen und übernehmen *)
	IF LC.RING_MODE THEN
		pos := LIMIT(1,pos,LC.SIZE - LV.COUNT + 1);
	ELSE
		IF LC.IDX > LV.COUNT THEN
			pos := LIMIT(1,pos,LC.IDX - LV.COUNT + 1);
		ELSE
			pos := 1;
		END_IF;
	END_IF;

	(* idxBasis berechnen *)
	base := LC.IDX - pos - LV.COUNT + 1;
	IF LC.RING_MODE THEN 
		(* Anzeige im Ringpuffermodus *)
		FOR count:= 1 TO LV.COUNT DO
			idx := base + count;
			IF idx < 1 THEN
				idx := idx + LC.SIZE;
			END_IF;
			LV.LINE_ARRAY[count] := idx;
		END_FOR;
	ELSE
		(* Anzeige im Normalmodus *)
		FOR count:= 1 TO LV.COUNT DO
			idx := base + count;
			IF idx < 1 THEN
				(* Leere Zeile ausgeben *)
				LV.LINE_ARRAY[count] := 0;
			ELSE
				LV.LINE_ARRAY[count] := idx;
			END_IF;
		END_FOR;
	END_IF;
END_IF;

(* revision history
ks	01. mai 2010	rev 1.0
	original version

ks	05. mai 2012	rev 1.1
	Fehler im Ringmodus

*)

END_FUNCTION_BLOCK

// POUs/NETWORK/MB_CLIENT
FUNCTION_BLOCK MB_CLIENT
VAR_IN_OUT
	IP_C : IP_C;
	S_BUF : NETWORK_BUFFER_SHORT;
	R_BUF : NETWORK_BUFFER_SHORT;
	DATA : ARRAY [0..255] OF WORD;
END_VAR
VAR_INPUT
	DATA_SIZE : INT;
	ENABLE : BOOL;
	UDP : BOOL;
	FC : INT;
	UNIT_ID : BYTE;
	R_ADDR : INT;
	R_POINTS : INT;
	R_DATA_ADR : INT;
	R_DATA_BITPOS : INT;
	W_ADDR : INT;
	W_POINTS : INT;
	W_DATA_ADR : INT;
	W_DATA_BITPOS : INT;
	DELAY : TIME;
END_VAR
VAR_OUTPUT
	ERROR : DWORD;
	BUSY : BOOL;
END_VAR
VAR
	ip_state : BYTE;
	ip_id : BYTE;
	ip_fifo : ip_fifo;
	mask : DWORD;
	w_tmp : WORD;
	idx1 : INT;
	idx2 : INT;
	stop : INT;
	i : INT;
	bit_pos : INT;
	w_mask : WORD;
	b_mask : BYTE;
	count : INT;
	state : INT;
	transaction_id : INT;
	response : INT;
	comp : INT;
	ton_1 : TON;
END_VAR

(*
version 1.2		20. oct. 2009
programmer 		ks
tested BY		ks

MB_CLIENT ermöglicht das Lesen/Schreiben von Daten über das Protokoll Modbus over Ethernet (OpenModbus)
*)

CASE state OF

00: (* Warten auf Delay-Time *)
	TON_1(IN:=ENABLE,PT:=DELAY);

	IF TON_1.Q OR DELAY = T#0s THEN
		TON_1(IN:=FALSE);
		state := 20;
		IP_STATE := BYTE#1; (* Anmelden *)
	END_IF;

20: (* Bei IP_Control anmelden *)
	IF IP_STATE = BYTE#3 THEN
		(* IP Datenverkehr einrichten *)
		IP_C.C_PORT := WORD#0; (* Port von IP_CONTROL verwenden *)
		IP_C.C_IP := DWORD#0; (* IP von IP_CONTROL verwenden *)
		IP_C.C_MODE := BOOL_TO_BYTE(UDP); (* Mode: 0=TCP+ACTIVE+IP , 1=UDP+ACTIVE+IP *)
		IP_C.TIME_RESET := TRUE; (* Zeitueberwachung rücksetzen *)
		IP_C.C_ENABLE := TRUE; (* Verbindungsaufbau freigeben *)
		IP_C.R_OBSERVE := TRUE; (* Empfangsueberwachung *)
		ERROR := DWORD#00; (* letzten Fehler rücksetzen *)

		CASE FC OF
		(******************************************************************)
		1..2: (* 0x01 Read Coil Status , 0x02 Read Input Status *)
			IF R_POINTS <= 2000 THEN
				w_tmp := INT_TO_WORD(R_ADDR);
				S_BUF.BUFFER[08] := WORD_TO_BYTE(SHR(w_tmp,8));
				S_BUF.BUFFER[09] := WORD_TO_BYTE(w_tmp);
				w_tmp := INT_TO_WORD(R_POINTS);
				S_BUF.BUFFER[10] := WORD_TO_BYTE(SHR(w_tmp,8));
				S_BUF.BUFFER[11] := WORD_TO_BYTE(w_tmp);
				S_BUF.SIZE := UINT#12;
				Response :=	WORD_TO_INT(SHR(INT_TO_WORD(R_POINTS + 7),3));
				comp := 7;
			ELSE
				ERROR := DWORD#2; (* ILLEGAL DATA ADDRESS *)
			END_IF;
		(******************************************************************)
		3..4: (* 0x03 Read Holding Registers , 0x04 Read Input Registers *)
			IF R_POINTS <= 125 THEN
				w_tmp := INT_TO_WORD(R_ADDR);
				S_BUF.BUFFER[08] := WORD_TO_BYTE(SHR(w_tmp,8));
				S_BUF.BUFFER[09] := WORD_TO_BYTE(w_tmp);
				w_tmp := INT_TO_WORD(R_POINTS);
				S_BUF.BUFFER[10] := WORD_TO_BYTE(SHR(w_tmp,8));
				S_BUF.BUFFER[11] := WORD_TO_BYTE(w_tmp);
				S_BUF.SIZE := UINT#12;
				Response :=	WORD_TO_INT(SHL(w_tmp,1));
				comp := 7;
			ELSE
				ERROR := DWORD#2; (* ILLEGAL DATA ADDRESS *)
			END_IF;
		(******************************************************************)
		5:	(* 0x05 Force Single Coil *)
			IF W_DATA_ADR <= DATA_SIZE THEN
				w_tmp := INT_TO_WORD(W_ADDR);
				S_BUF.BUFFER[08] := WORD_TO_BYTE(SHR(w_tmp,8));
				S_BUF.BUFFER[09] := WORD_TO_BYTE(w_tmp);
				S_BUF.BUFFER[10] := SEL((DATA[W_DATA_ADR] AND SHL(WORD#1,W_DATA_BITPOS))>WORD#00,BYTE#16#00,BYTE#16#FF);
				S_BUF.BUFFER[11] := BYTE#00;
				S_BUF.SIZE := UINT#12;
				Response := 3;
				comp := 11;
			ELSE
				ERROR := DWORD#2; (* ILLEGAL DATA ADDRESS *)
			END_IF;
		(******************************************************************)
		6:	(* 0x06 Preset Single Register *)
			IF W_DATA_ADR <= DATA_SIZE THEN
				w_tmp := INT_TO_WORD(W_ADDR);
				S_BUF.BUFFER[08] := WORD_TO_BYTE(SHR(w_tmp,8));
				S_BUF.BUFFER[09] := WORD_TO_BYTE(w_tmp);
				w_tmp := DATA[W_DATA_ADR];
				S_BUF.BUFFER[10] := WORD_TO_BYTE(SHR(w_tmp,8));
				S_BUF.BUFFER[11] := WORD_TO_BYTE(w_tmp);
				S_BUF.SIZE := UINT#12;
				Response := 3;
				comp := 11;
			ELSE
				ERROR := DWORD#2; (* ILLEGAL DATA ADDRESS *)
			END_IF;
		(******************************************************************)
		15:	(* 0x0F Force Multiple Coils *)
			IF (WORD_TO_INT(SHR(INT_TO_WORD(WORD_TO_INT(SHL(INT_TO_WORD(W_DATA_ADR),4)) + W_POINTS + W_DATA_BITPOS + 15),4)) <= DATA_SIZE) AND W_POINTS <= 1968 THEN
				w_tmp := INT_TO_WORD(W_ADDR);
				S_BUF.BUFFER[08] := WORD_TO_BYTE(SHR(w_tmp,8));
				S_BUF.BUFFER[09] := WORD_TO_BYTE(w_tmp);
				w_tmp := INT_TO_WORD(W_POINTS);
				S_BUF.BUFFER[10] := WORD_TO_BYTE(SHR(w_tmp,8));
				S_BUF.BUFFER[11] := WORD_TO_BYTE(w_tmp);
				S_BUF.BUFFER[12] := WORD_TO_BYTE(SHR(INT_TO_WORD(W_POINTS + 7),3));

				w_mask := SHL(WORD#1,W_DATA_BITPOS);
				bit_pos := 0;
				w_tmp := WORD#00;
				idx1 := 12;
				idx2 := W_DATA_ADR;
				FOR i := 1 TO W_POINTS DO
					w_tmp :=OSCAT_BASIC.BIT_LOAD_W(w_tmp,(DATA[idx2] AND w_mask) > WORD#0,bit_pos);
					bit_pos := bit_pos + 1;
					IF bit_pos > 7 OR i=W_POINTS THEN
						bit_pos := 0;
						idx1 := idx1 + 1;
						S_BUF.BUFFER[idx1] := WORD_TO_BYTE(w_tmp);
						w_tmp := WORD#0;
					END_IF;
					w_mask := ROL(w_mask,1);
					IF w_mask = WORD#1 THEN
						idx2 := idx2 +1;
					END_IF;
				END_FOR;
				S_BUF.SIZE := INT_TO_UINT(idx1 + 1);
				Response := 3;
				comp := 11;
			ELSE
				ERROR := DWORD#2; (* ILLEGAL DATA ADDRESS *)
			END_IF;
		(******************************************************************)
		16:	(* 0x10 Write Multiple Registers *)
			IF W_DATA_ADR + W_POINTS <= DATA_SIZE AND W_POINTS <= 123 THEN
				w_tmp := INT_TO_WORD(W_ADDR);
				S_BUF.BUFFER[08] := WORD_TO_BYTE(SHR(w_tmp,8));
				S_BUF.BUFFER[09] := WORD_TO_BYTE(w_tmp);
				w_tmp := INT_TO_WORD(W_POINTS);
				S_BUF.BUFFER[10] := WORD_TO_BYTE(SHR(w_tmp,8));
				S_BUF.BUFFER[11] := WORD_TO_BYTE(w_tmp);
				S_BUF.BUFFER[12] := SHL(S_BUF.BUFFER[11],1);
			
				idx1 := 11;
				count := W_DATA_ADR + W_POINTS - 1;
				FOR i := W_DATA_ADR TO count DO
					idx1 := idx1 + 2;
					idx2 := idx1 + 1; (* zweiter index für pcworx notwendig ! *)
					w_tmp := DATA[i];
					S_BUF.BUFFER[idx1] := WORD_TO_BYTE(SHR(w_tmp,8));
					S_BUF.BUFFER[idx2] := WORD_TO_BYTE(w_tmp);
				END_FOR;

				S_BUF.SIZE := INT_TO_UINT(idx2 + 1);
				Response := 3;
				comp := 11;
			ELSE
				ERROR := DWORD#2; (* ILLEGAL DATA ADDRESS *)
			END_IF;
		(******************************************************************)
		22:	(* 0x16 Mask Write Register *)
			IF W_DATA_ADR + 2 <= DATA_SIZE THEN
				w_tmp := INT_TO_WORD(W_ADDR);
				S_BUF.BUFFER[08] := WORD_TO_BYTE(SHR(w_tmp,8));
				S_BUF.BUFFER[09] := WORD_TO_BYTE(w_tmp);
				idx1 := W_DATA_ADR;
				w_tmp := DATA[idx1];
				S_BUF.BUFFER[10] := WORD_TO_BYTE(SHR(w_tmp,8));
				S_BUF.BUFFER[11] := WORD_TO_BYTE(w_tmp);
				idx1 := idx1 +1;
				w_tmp := DATA[idx1];
				S_BUF.BUFFER[12] := WORD_TO_BYTE(SHR(w_tmp,8));
				S_BUF.BUFFER[13] := WORD_TO_BYTE(w_tmp);

				S_BUF.SIZE := UINT#14;
				Response := 5;
				comp := 13;
			ELSE
				ERROR := DWORD#2; (* ILLEGAL DATA ADDRESS *)
			END_IF;
		(******************************************************************)
		23:	(* 0x17 Read/Write Multible Registers *)
			IF W_DATA_ADR + W_POINTS <= DATA_SIZE AND W_POINTS <= 121 AND R_POINTS <= 125 THEN
				idx1 := 15;
				count := W_DATA_ADR + W_POINTS - 1;
				FOR i := W_DATA_ADR TO count DO
					idx1 := idx1 + 2;
					idx2 := idx1 + 1; (* zweiter index für pcworx notwendig ! *)
					w_tmp := DATA[i];
					S_BUF.BUFFER[idx1] := WORD_TO_BYTE(SHR(w_tmp,8));
					S_BUF.BUFFER[idx2] := WORD_TO_BYTE(w_tmp);
				END_FOR;

				(* WRITE *)
				w_tmp := INT_TO_WORD(W_ADDR);
				S_BUF.BUFFER[12] := WORD_TO_BYTE(SHR(w_tmp,8));
				S_BUF.BUFFER[13] := WORD_TO_BYTE(w_tmp);
				w_tmp := INT_TO_WORD(W_POINTS);
				S_BUF.BUFFER[14] := WORD_TO_BYTE(SHR(w_tmp,8));
				S_BUF.BUFFER[15] := WORD_TO_BYTE(w_tmp);
				S_BUF.BUFFER[16] := SHL(S_BUF.BUFFER[15],1);

				(* READ *)
				w_tmp := INT_TO_WORD(R_ADDR);
				S_BUF.BUFFER[08] := WORD_TO_BYTE(SHR(w_tmp,8));
				S_BUF.BUFFER[09] := WORD_TO_BYTE(w_tmp);
				w_tmp := INT_TO_WORD(R_POINTS);
				S_BUF.BUFFER[10] := WORD_TO_BYTE(SHR(w_tmp,8));
				S_BUF.BUFFER[11] := WORD_TO_BYTE(w_tmp);

				S_BUF.SIZE := INT_TO_UINT(idx2 + 1);
				Response := WORD_TO_INT(SHL(w_tmp,1));
				comp := 7;
			ELSE
				ERROR := DWORD#2; (* ILLEGAL DATA ADDRESS *)
			END_IF;
		(******************************************************************)

		ELSE
			ERROR := DWORD#00000001; (* ILLEGAL FUNCTION *)
		END_CASE;

		(* Daten senden *)
		IF ERROR = DWORD#00 THEN
			Transaction_ID := Transaction_ID + 1;
			w_tmp := UINT_TO_WORD(S_BUF.SIZE - UINT#6);
			(* ---- H E A D E R --------------------------------------------------------------- *)
			S_BUF.BUFFER[0] := IP_ID; (* TRANSACTION-ID HI-Byte *)
			S_BUF.BUFFER[1] := INT_TO_BYTE(Transaction_ID); (* TRANSACTION-ID LO-Byte *)
			S_BUF.BUFFER[2] := BYTE#00; (* PROTOKOLL-ID HI-Byte *)
			S_BUF.BUFFER[3] := BYTE#00; (* PROTOKOLL-ID LO-Byte *)
			S_BUF.BUFFER[4] := WORD_TO_BYTE(SHR(w_tmp,8)); (* Laenge HI-Byte *)
			S_BUF.BUFFER[5] := WORD_TO_BYTE(w_tmp); (* Laenge LO-Byte *)
			S_BUF.BUFFER[6] := UNIT_ID; (* UNIT *)
			S_BUF.BUFFER[7] := INT_TO_BYTE(FC); (* FUNCTION-CODE *)
			(*----- END OF HEADER --------------------------------------------------------------*)
			R_BUF.SIZE := UINT#0; (* Empfangsbuffer löschen *)
			state := 30; (* wait for response *)
		ELSE
			IP_STATE := BYTE#4; (* Abmelden *)
			state := 00;
		END_IF;
	END_IF;

30: (* response *)
	IF IP_C.ERROR <> DWORD#00 THEN
		ERROR := IP_C.ERROR;
		IP_STATE := BYTE#4; (* Abmelden *)
		state := 00;
	ELSIF S_BUF.SIZE = UINT#0 AND R_BUF.SIZE > UINT#0 THEN
		(* erwartete länge in sendebuffer nachträglich eintragen um vergleich zu ermöglichen *)
		w_tmp := INT_TO_WORD(Response + 3);
		S_BUF.BUFFER[4] := WORD_TO_BYTE(SHR(w_tmp,8));
		S_BUF.BUFFER[5] := WORD_TO_BYTE(w_tmp);

		FOR i := 0 TO comp DO
			IF S_BUF.BUFFER[i] <> R_BUF.BUFFER[i] THEN EXIT; END_IF;
		END_FOR;

		IF R_BUF.SIZE >= UINT#9 AND R_BUF.BUFFER[7] > BYTE#128 THEN  (* Bit 7 = Error Message *)
			ERROR := BYTE_TO_DWORD(R_BUF.BUFFER[8]);
			IP_STATE := BYTE#4; (* Abmelden *)
			state := 00;
		ELSIF R_BUF.SIZE = INT_TO_UINT(Response + 9) AND i > comp THEN
			mask := SHL(DWORD#1,FC);
			(* READ_COILS, READ_INPUT_DISCRETES *)
			IF (mask AND DWORD#2#00000000_00000000_00000000_00000110) > DWORD#0 THEN (* FC 1,2 *)
				IF WORD_TO_INT(SHR(INT_TO_WORD(WORD_TO_INT(SHL(INT_TO_WORD(R_DATA_ADR),4)) + R_POINTS + R_DATA_BITPOS + 15),4)) <= DATA_SIZE THEN
					b_mask := BYTE#1;
					idx1 := 09;
					idx2 := R_DATA_ADR;
					bit_pos := R_DATA_BITPOS;
					FOR i := 1 TO R_POINTS DO
						DATA[idx2]:=OSCAT_BASIC.BIT_LOAD_W(DATA[idx2],(R_BUF.BUFFER[idx1] AND b_mask) > BYTE#0,bit_pos);
						bit_pos := bit_pos + 1;
						IF bit_pos > 15 THEN
							idx2 := idx2 + 1;
							bit_pos := 0;
						END_IF;
						b_mask := ROL(b_mask,1);
						IF b_mask = BYTE#1 THEN
							idx1 := idx1 + 1;
						END_IF;
					END_FOR;
				ELSE
					ERROR := DWORD#2; (* ILLEGAL DATA ADDRESS *)
				END_IF;

			(* READ_MULTIPLE_REGISTERS, READ_INPUT_REGISTERS, READ_WRITE_REGISTERS *)
			ELSIF (mask AND DWORD#2#00000000_10000000_00000000_00011000) > DWORD#0 THEN (* FC 3,4,23 *)
				IF R_DATA_ADR + R_POINTS <= DATA_SIZE THEN
					stop := R_DATA_ADR + R_POINTS -1 ;
					idx1 := 07;
					FOR i := R_DATA_ADR TO stop DO
						idx1 := idx1 + 2;
						idx2 := idx1 + 1;
						DATA[i] := OSCAT_BASIC.WORD_OF_BYTE(R_BUF.BUFFER[idx1],R_BUF.BUFFER[idx2]);
					END_FOR;
				ELSE
					ERROR := DWORD#2; (* ILLEGAL DATA ADDRESS *)
				END_IF;
			ELSIF (mask AND DWORD#2#11111111_00111110_01111111_10000001) > DWORD#0 THEN (* ILLEGAL FUNCTION CODE ? *)
				ERROR := DWORD#1; (* ILLEGAL FUNCTION *)
			END_IF;
		ELSE
			ERROR := DWORD#3; (* ILLEGAL DATA VALUE *)
		END_IF;

		IP_STATE := BYTE#4; (* Abmelden *)
		state := 00;
		R_BUF.SIZE := UINT#0;

	END_IF;

END_CASE;

(* IP_FIFO *)
IP_FIFO(FIFO:=IP_C.FIFO,STATE:=IP_STATE,ID:=IP_ID);
BUSY := IP_STATE = BYTE#3;

(* revision history
ks	05. jan. 2009	rev 1.0
	original version

ks	28. jan. 2009	rev 1.1
	network_buffer_short verwendet  

ks	20. oct. 2009	rev 1.2
Networkbuffer und Buffer-funktionen auf Basis 0

*)

END_FUNCTION_BLOCK

// POUs/DEMO/MB_CLIENT_DEMO
PROGRAM MB_CLIENT_DEMO
VAR
	IP_CONTROL2_1: IP_CONTROL2;
	MB_CLIENT_1: MB_CLIENT;
	IP_C: IP_C;
	S_BUF: NETWORK_BUFFER_SHORT;
	R_BUF: NETWORK_BUFFER_SHORT;
	DATA: ARRAY [0..255] OF WORD;
	W_DATA_BITPOS: INT;
	W_DATA_ADR: INT;
	W_POINTS: INT;
	W_ADDR: INT;
	R_DATA_BITPOS: INT;
	R_DATA_ADR: INT;
	R_POINTS: INT;
	R_ADDR: INT;
	FC: INT;
	ENABLE: BOOL;
END_VAR
VAR // added by the converter: edge detectors and wires of the graphical bodies
    _w1 : ANY;
END_VAR

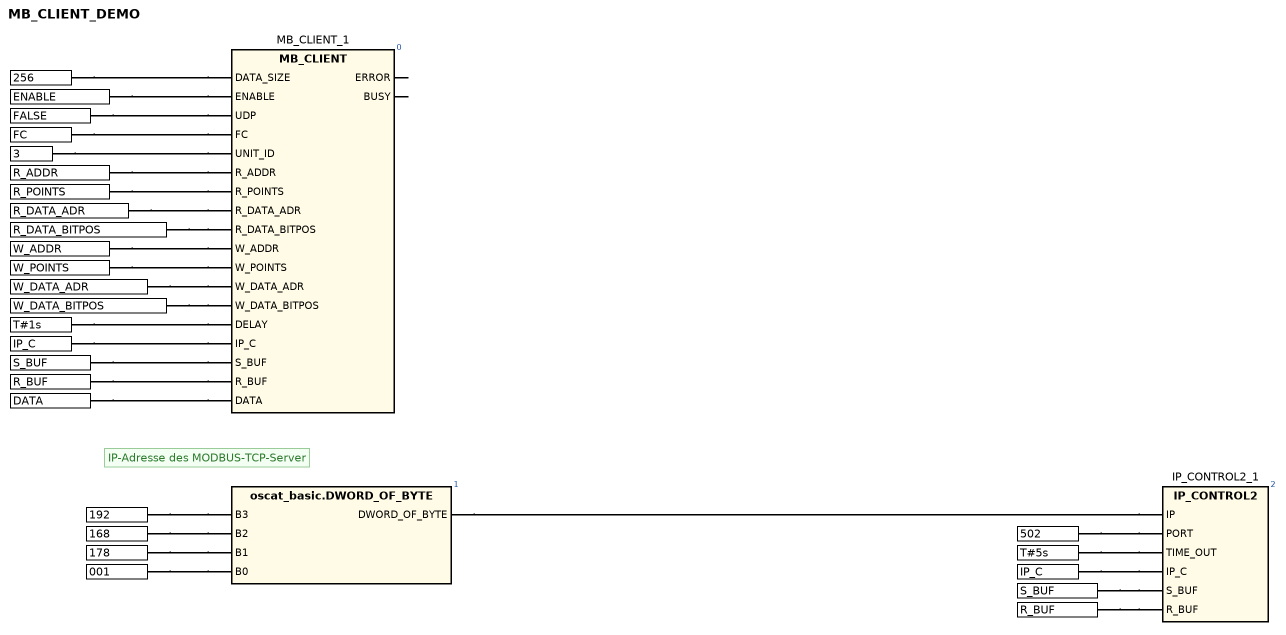
MB_CLIENT_1(
    DATA_SIZE := 256,
    ENABLE := ENABLE,
    UDP := FALSE,
    FC := FC,
    UNIT_ID := 3,
    R_ADDR := R_ADDR,
    R_POINTS := R_POINTS,
    R_DATA_ADR := R_DATA_ADR,
    R_DATA_BITPOS := R_DATA_BITPOS,
    W_ADDR := W_ADDR,
    W_POINTS := W_POINTS,
    W_DATA_ADR := W_DATA_ADR,
    W_DATA_BITPOS := W_DATA_BITPOS,
    DELAY := T#1s,
    IP_C := IP_C,
    S_BUF := S_BUF,
    R_BUF := R_BUF,
    DATA := DATA); // MB_CLIENT
// IP-Adresse des MODBUS-TCP-Server
_w1 := oscat_basic.DWORD_OF_BYTE(B3 := 192, B2 := 168, B1 := 178, B0 := 001);
IP_CONTROL2_1(IP := _w1, PORT := 502, TIME_OUT := T#5s, IP_C := IP_C, S_BUF := S_BUF, R_BUF := R_BUF); // IP_CONTROL2

END_PROGRAM

// POUs/NETWORK/MB_SERVER
FUNCTION_BLOCK MB_SERVER
VAR_IN_OUT
	IP_C : IP_C;
	S_BUF : NETWORK_BUFFER_SHORT;
	R_BUF : NETWORK_BUFFER_SHORT;
	VMAP : ARRAY [1..10] OF VMAP_DATA;
	DATA : ARRAY [0..255] OF WORD;
END_VAR
VAR_INPUT
	DATA_SIZE : INT;
	ENABLE : BOOL;
	UDP : BOOL;
END_VAR
VAR_OUTPUT
	ERROR : DWORD;
END_VAR
VAR
	MB_VMAP : MB_VMAP;
	adr1 : INT;
	adr2 : INT;
	points : INT;
	points2 : INT;
	coils : BYTE;
	mask : BYTE;
	idx1 : INT;
	idx2 : INT;
	bit_pos : INT;
	count : INT;
	fc : INT;
	i : INT;
	state : INT;
	ip_state : BYTE;
	ip_id : BYTE;
	IP_FIFO : IP_FIFO;
	w_tmp : WORD;
	last_cycle : TIME;
	tx : TIME;
	t : TON;
	ip_error : BOOL;
END_VAR

(*

version 1.4		05. may. 2012
programmer 		ks
tested by		ks

MB_SERVER ermöglicht das Lesen/Schreiben von Daten durch ein Remote-Device mittels Modbus over Ethernet (OpenModbus)

*)

(* read system time *)
tx := DWORD_TO_TIME(OSCAT_BASIC.T_PLC_MS());

FOR i := 1 TO 10 DO
	IF VMAP[i].TIME_OUT > T#0s THEN
		VMAP[i].TIME_OUT := VMAP[i].TIME_OUT + tx - last_cycle;
	END_IF;
END_FOR;
last_cycle := tx;
ip_error := IP_C.ERROR > DWORD#0;

CASE state OF
00: (* Warten auf Freigabe *)
	IF ENABLE THEN
		state := 10;
		ip_state := BYTE#1; (* Anmelden *)
	END_IF;

10: (* Bei IP_Control anmelden und auf freigabe warten *)
	IF ip_state = BYTE#3 THEN

		(* IP Datenverkehr einrichten *)
		IP_C.C_PORT := WORD#0; (* Port von IP_CONTROL verwenden *)
		IP_C.C_IP := DWORD#0; (* IP von IP_CONTROL verwenden *)
		IP_C.C_MODE := SEL(UDP,BYTE#4,BYTE#5); (* Mode: 4=TCP+PASSIV+PORT , 5=UDP+PASSIV+PORT *)
		IP_C.TIME_RESET := TRUE; (* Zeitueberwachung rücksetzen *)
		IP_C.C_ENABLE := TRUE; (* Verbindungsaufbau freigeben *)
		IP_C.R_OBSERVE := TRUE; (* keine Empfangsueberwachung *)
		state := 20;
	END_IF;

20:	IF NOT ip_error THEN
		IF S_BUF.SIZE = UINT#0 AND R_BUF.SIZE > UINT#6 THEN	(* Datensenden nicht aktiv und Daten wurden empfangen *)
			IF  R_BUF.SIZE = WORD_TO_UINT(OSCAT_BASIC.WORD_OF_BYTE(R_BUF.BUFFER[4],R_BUF.BUFFER[5])) + UINT#6 THEN (* gültige Datenlänge *)
				ERROR := DWORD#00; (* Error löschen *)

				(* Header kopieren *)
				FOR i := 0 TO 13 DO
					S_BUF.BUFFER[i] := R_BUF.BUFFER[i];
				END_FOR;
				fc := BYTE_TO_INT(R_BUF.BUFFER[7]);
				adr1 := WORD_TO_INT(OSCAT_BASIC.WORD_OF_BYTE(R_BUF.BUFFER[8],R_BUF.BUFFER[9]));
				points := WORD_TO_INT(OSCAT_BASIC.WORD_OF_BYTE(R_BUF.BUFFER[10],R_BUF.BUFFER[11]));

				(* Virtual Address *)
				MB_VMAP(VMAP:=VMAP,FC:=fc,V_ADR:=adr1,V_CNT:=points,SIZE:=DATA_SIZE);
				adr1:=MB_VMAP.P_ADR;
				bit_pos:=MB_VMAP.P_BIT;
				ERROR:=BYTE_TO_DWORD(MB_VMAP.ERROR);

				IF ERROR = DWORD#0 THEN
					CASE fc OF
					(*---------------------------------------------*)
					1..2 : (* Read Coil Status / Read Input Status *)
						count := 9; (* erstes Datenbyte *)
						coils := BYTE#0;
						mask := BYTE#1;
						FOR i := 1 TO points DO
							IF mask = BYTE#0 THEN
								mask := BYTE#1;
								S_BUF.BUFFER[count] := coils;
								coils := BYTE#0;
								count := count + 1;
							END_IF;
							IF (DATA[adr1] AND SHL(WORD#1,bit_pos)) > WORD#0 THEN
								coils := coils OR mask;
							END_IF;
	
							bit_Pos := bit_Pos + 1;
							IF bit_pos > 15 THEN
								ADR1 := ADR1 + 1;
								bit_pos := 0;
							END_IF;
	
							mask := SHL(mask,1);
						END_FOR;
						S_BUF.BUFFER[Count] := coils;
	
						S_BUF.BUFFER[8] := INT_TO_BYTE(count - 8); (* Bytecount *)
						S_BUF.SIZE := INT_TO_UINT(count + 1);
	
					(*--------------------------------------------------*)
					3..4 : (* Read Holding Registers / Read Input Registers *)
						idx1 := 07;
						count := adr1 + points - 1;
						FOR i := adr1 TO count DO
							idx1 := idx1 + 2;
							idx2 := idx1 + 1; (* zweiter index für pcworx notwendig ! *)
							w_tmp := DATA[i];
							S_BUF.BUFFER[idx1] := WORD_TO_BYTE(SHR(w_tmp,8));
							S_BUF.BUFFER[idx2] := WORD_TO_BYTE(w_tmp);
						END_FOR;
						S_BUF.BUFFER[8] := SHL(INT_TO_BYTE(points),1); (* Anzahl Register in Bytes *)
						S_BUF.SIZE := INT_TO_UINT(idx2 + 1);
					(*--------------------------------------------------*)
					5 : (* Force Single Coil *)
						DATA[adr1]:=OSCAT_BASIC.BIT_LOAD_W(DATA[adr1],R_BUF.BUFFER[10] > BYTE#0,bit_pos);
						S_BUF.SIZE := UINT#12;
					(*--------------------------------------------------*)
					6 : (* Preset Single Register *)
						DATA[adr1] := OSCAT_BASIC.WORD_OF_BYTE(R_BUF.BUFFER[10],R_BUF.BUFFER[11]);
						S_BUF.SIZE := UINT#12;
					(*--------------------------------------------------*)
					15 : (* Force Multible Coils *)
						mask := BYTE#1;
						idx1 := 13;
						FOR i := 1 TO points DO
							DATA[adr1]:=OSCAT_BASIC.BIT_LOAD_W(DATA[adr1],(R_BUF.BUFFER[idx1] AND mask) > BYTE#0,bit_pos);
							bit_pos := bit_pos + 1;
							IF bit_pos > 15 THEN
								adr1:= adr1 + 1;
								bit_pos := 0;
							END_IF;
							mask := ROL(mask,1);
							IF mask = BYTE#1 THEN
								idx1 := idx1 +1;
							END_IF;
						END_FOR;
						S_BUF.SIZE := UINT#12;
					(*--------------------------------------------------*)
					16 : (* Preset Multiple Registers	*)
						idx1 := 11;
						count := adr1 + points - 1;
						FOR i := adr1 TO Count DO
							idx1 := idx1 + 2;
	 						idx2 := idx1 + 1;
							Data[i] := OSCAT_BASIC.WORD_OF_BYTE(R_BUF.BUFFER[idx1],R_BUF.BUFFER[idx2]);
						END_FOR;
						S_BUF.SIZE := UINT#12;
					(*--------------------------------------------------*)
					22 : (* Mask Write Register *)
						w_tmp := OSCAT_BASIC.WORD_OF_BYTE(R_BUF.BUFFER[10],R_BUF.BUFFER[11]); (* and mask *)
						DATA[adr1] := (DATA[adr1] AND w_tmp) OR (OSCAT_BASIC.WORD_OF_BYTE(R_BUF.BUFFER[12],R_BUF.BUFFER[13]) AND (NOT w_tmp));
						S_BUF.SIZE := UINT#14;
					(*--------------------------------------------------*)
					23 : (* Read / Write Registers	*)
						(*--- Write-Register -----------------------------------*)
						adr2 := WORD_TO_INT(OSCAT_BASIC.WORD_OF_BYTE(R_BUF.BUFFER[12],R_BUF.BUFFER[13]));
						points2 := WORD_TO_INT(OSCAT_BASIC.WORD_OF_BYTE(R_BUF.BUFFER[14],R_BUF.BUFFER[15]));

						(* Virtual Address Write Register *)
						MB_VMAP(VMAP:=VMAP,FC:=16,V_ADR:=adr2,V_CNT:=points2,SIZE:=DATA_SIZE);
						adr2:=MB_VMAP.P_ADR;
						ERROR:=BYTE_TO_DWORD(MB_VMAP.ERROR);
	
						IF ERROR = DWORD#0 THEN
							idx1 := 15;
							count := adr2 + points2 - 1;
							FOR i := adr2 TO count DO
								idx1 := idx1 + 2;
	 							idx2 := idx1 + 1; (* zweiter index für pcworx notwendig ! *)
								Data[i] := OSCAT_BASIC.WORD_OF_BYTE(R_BUF.BUFFER[idx1],R_BUF.BUFFER[idx2]);
							END_FOR;
	
							(*--- Read-Register -----------------------------------*)
							idx1 := 07;
							count := adr1 + points - 1;
							FOR i := adr1 TO count DO
								idx1 := idx1 + 2;
								idx2 := idx1 + 1; (* zweiter index für pcworx notwendig ! *)
								w_tmp := DATA[i];
								S_BUF.BUFFER[idx1] := WORD_TO_BYTE(SHR(w_tmp,8));
								S_BUF.BUFFER[idx2] := WORD_TO_BYTE(w_tmp);
							END_FOR;
							S_BUF.BUFFER[8] := SHL(INT_TO_BYTE(points),1); (* Anzahl Register in Bytes *)
							S_BUF.SIZE := INT_TO_UINT(idx2 + 1);
	
						END_IF;
	
					(*--------------------------------------------------*)
					ELSE
						ERROR := DWORD#01; (* ILLEGAL FUNCTION *)
					END_CASE;
				END_IF;
			END_IF;
	
			IF ERROR > DWORD#0 THEN
				S_BUF.BUFFER[7] := S_BUF.BUFFER[7] OR BYTE#2#1000_0000; (* Fehlerbit setzen *)
				S_BUF.BUFFER[8] := DWORD_TO_BYTE(ERROR);
				S_BUF.SIZE := UINT#9;
			END_IF;
	
			S_BUF.BUFFER[4] := BYTE#0; (* high Byte *)
			S_BUF.BUFFER[5] := UINT_TO_BYTE(S_BUF.SIZE - UINT#6); (* Längenfeld eintragen - nur low byte *)
	
		END_IF;
	ELSE
		ERROR := IP_C.ERROR;
	END_IF;

	t(IN:= ip_error, PT:=T#2s);
	IF t.Q THEN
		IP_C.TIME_RESET := TRUE; (* Error Reset *)
	END_IF;

	R_BUF.SIZE := UINT#0; (* Empfangsdaten zerstören *)

	IF ENABLE = FALSE OR t.Q THEN
	    ip_state := BYTE#4; (* Abmelden *)
		state := 00;
		IP_C.C_ENABLE := FALSE;
	END_IF;
END_CASE;

(* IP_FIFO *)
IP_FIFO(FIFO:=IP_C.FIFO,STATE:=ip_state,ID:=ip_id);

(* revision history
ks	05. jan. 2009	rev 1.0
	original version

ks	28. jan. 2009	rev 1.1
	network_buffer_short verwendet  

ks	20. oct. 2009	rev 1.2
	change lokal-var adr to adr1,Networkbuffer und Buffer-funktionen auf Basis 0

ks	17. may. 2011	rev 1.3
	automatischer re-connect

ks	05. may. 2012	rev 1.4
	timeoutüberwachung für re-connect
*)

END_FUNCTION_BLOCK

// POUs/NETWORK/MB_VMAP
FUNCTION_BLOCK MB_VMAP
VAR_IN_OUT
	VMAP :  ARRAY [1..10] OF VMAP_DATA;
END_VAR
VAR_INPUT
	FC : INT;
	V_ADR : INT;
	V_CNT : INT;
	SIZE : INT;
END_VAR
VAR_OUTPUT
	P_ADR : INT;
	P_BIT : INT;
	ERROR : BYTE;
END_VAR
VAR
	i : INT;
	vopt : DWORD;
	vadr : INT;
	padr : INT;
	mask : DWORD;
	vsize : INT;
	w_tmp : WORD;
	i_tmp : INT;
	init : BOOL;
END_VAR

(*
version 1.1		20. oct. 2009
programmer 		ks
tested by		ks

MB_VMAP Virtuelles Adress-Mapping für MB_SERVER
*)

IF init = FALSE THEN
	init := TRUE;
	IF VMAP[1].FC = DWORD#0 THEN
		VMAP[1].FC := DWORD#16#FFFF_FFFF;
		VMAP[1].V_ADR := 0;
		VMAP[1].V_SIZE := 256;
		VMAP[1].P_ADR := 0;
	END_IF;
END_IF;

ERROR := BYTE#02; (* ILLEGAL DATA ADDRESS *)
mask := SHL(DWORD#1,FC);

IF (mask AND DWORD#2#00000000_01000000_00000000_01100000) <> DWORD#0 THEN (* FC 5,6,22 *)
	V_CNT := 1;
ELSIF V_CNT = 0 THEN
	RETURN;
END_IF;

FOR i := 1 TO 10 DO
	vopt := VMAP[i].FC; 
	IF (vopt AND mask) <> DWORD#0 THEN
		vadr := VMAP[i].V_ADR;
		vsize := VMAP[i].V_SIZE;
		padr := VMAP[i].P_ADR;

		IF (mask AND DWORD#2#00000000_00000000_10000000_00100110) <> DWORD#0 THEN (* FC 1,2,5,15 für Bit-Access *)
			i_tmp := WORD_TO_INT(SHR(INT_TO_WORD(V_ADR + V_CNT -1),4))+1;
			IF i_tmp <= SIZE AND i_tmp <= vsize THEN
				w_tmp := INT_TO_WORD(V_ADR);
				P_ADR := WORD_TO_INT(SHR(w_tmp,4)) + padr; 
				P_BIT := WORD_TO_INT(w_tmp AND WORD#16#000F);
				ERROR := BYTE#0;
				EXIT;
			END_IF;
		ELSIF (mask AND DWORD#2#00000000_11000001_00000000_01011000) <> DWORD#0 THEN (* FC 3,4,6,16,22,23 für Register-Access *)
			IF V_ADR >= vadr AND V_ADR + V_CNT <= vadr + vsize THEN (* gültiger virtueller bereich *)
				P_ADR := V_ADR - vadr + padr; (* reale Adresse berechnen *)
				IF P_ADR + V_CNT <= SIZE THEN (* bereichsueberschreitung ? *)
					ERROR := BYTE#0;
					EXIT;
				END_IF;
			END_IF;
		ELSE
			ERROR := BYTE#01; (* ILLEGAL FUNCTION *)
			RETURN;
		END_IF;
	END_IF;
END_FOR;

IF ERROR = BYTE#0 THEN
	IF (mask AND DWORD#2#00000000_11000001_10000000_01100000) <> DWORD#0 THEN (* FC 5,6,15,16,22,23 Schreib-zugriff *)
		VMAP[i].TIME_OUT := T#1ms;
	END_IF;
END_IF;

(* revision history
ks	05. jan. 2009	rev 1.0
	original version

ks	20. oct. 2009	rev 1.1
	fehlerkorrektur in bitmaske

*)

END_FUNCTION_BLOCK

// POUs/NETWORK/MB_SERVER_1
FUNCTION_BLOCK MB_SERVER_1
VAR_IN_OUT
	IP_C : IP_C;
	S_BUF : NETWORK_BUFFER_SHORT;
	R_BUF : NETWORK_BUFFER_SHORT;
	VMAP : ARRAY [1..10] OF VMAP_DATA;
	DATA : ARRAY [0..255] OF WORD;
END_VAR
VAR_INPUT
	DATA_SIZE : INT;
	ENABLE : BOOL;
	UDP : BOOL;
END_VAR
VAR_OUTPUT
	ERROR : DWORD;
END_VAR
VAR
	MB_VMAP : MB_VMAP;
	adr1 : INT;
	adr2 : INT;
	points : INT;
	points2 : INT;
	coils : BYTE;
	mask : BYTE;
	idx1 : INT;
	idx2 : INT;
	bit_pos : INT;
	count : INT;
	fc : INT;
	i : INT;
	state : INT;
	ip_state : BYTE;
	ip_id : BYTE;
	IP_FIFO : IP_FIFO;
	w_tmp : WORD;
	last_cycle : TIME;
	tx : TIME;
	t : TON;
	ip_error : BOOL;
END_VAR

(*

version 1.3		17. may. 2011
programmer 		ks
tested by			ks

MB_SERVER ermöglicht das Lesen/Schreiben von Daten durch ein Remote-Device mittels Modbus over Ethernet (OpenModbus)

*)

(* read system time *)
tx := DWORD_TO_TIME(OSCAT_BASIC.T_PLC_MS());

FOR i := 1 TO 10 DO
	IF VMAP[i].TIME_OUT > T#0s THEN
		VMAP[i].TIME_OUT := VMAP[i].TIME_OUT + tx - last_cycle;
	END_IF;
END_FOR;
last_cycle := tx;
ip_error := IP_C.ERROR > DWORD#0;

CASE state OF
00: (* Warten auf Freigabe *)
	IF ENABLE THEN
		state := 10;
		ip_state := BYTE#1; (* Anmelden *)
	END_IF;

10: (* Bei IP_Control anmelden und auf freigabe warten *)
	IF ip_state = BYTE#3 THEN

		(* IP Datenverkehr einrichten *)
		IP_C.C_PORT := WORD#0; (* Port von IP_CONTROL verwenden *)
		IP_C.C_IP := DWORD#0; (* IP von IP_CONTROL verwenden *)
		IP_C.C_MODE := SEL(UDP,BYTE#4,BYTE#5); (* Mode: 4=TCP+PASSIV+PORT , 5=UDP+PASSIV+PORT *)
		IP_C.TIME_RESET := TRUE; (* Zeitueberwachung rücksetzen *)
		IP_C.C_ENABLE := TRUE; (* Verbindungsaufbau freigeben *)
		IP_C.R_OBSERVE := FALSE; (* keine Empfangsueberwachung *)
		state := 20;
	END_IF;

20:	IF NOT ip_error THEN
		IF S_BUF.SIZE = UINT#0 AND R_BUF.SIZE > UINT#6 THEN	(* Datensenden nicht aktiv und Daten wurden empfangen *)
			IF  R_BUF.SIZE = WORD_TO_UINT(OSCAT_BASIC.WORD_OF_BYTE(R_BUF.BUFFER[4],R_BUF.BUFFER[5])) + UINT#6 THEN (* gültige Datenlänge *)
				ERROR := DWORD#00; (* Error löschen *)
	
				(* Header kopieren *)
				FOR i := 0 TO 13 DO
					S_BUF.BUFFER[i] := R_BUF.BUFFER[i];
				END_FOR;
				fc := BYTE_TO_INT(R_BUF.BUFFER[7]);
				adr1 := WORD_TO_INT(OSCAT_BASIC.WORD_OF_BYTE(R_BUF.BUFFER[8],R_BUF.BUFFER[9]));
				points := WORD_TO_INT(OSCAT_BASIC.WORD_OF_BYTE(R_BUF.BUFFER[10],R_BUF.BUFFER[11]));
	
				(* Virtual Address *)
				MB_VMAP(VMAP:=VMAP,FC:=fc,V_ADR:=adr1,V_CNT:=points,SIZE:=DATA_SIZE);
				adr1:=MB_VMAP.P_ADR;
				bit_pos:=MB_VMAP.P_BIT;
				ERROR:=BYTE_TO_DWORD(MB_VMAP.ERROR);
	
				IF ERROR = DWORD#0 THEN
					CASE fc OF
					(*---------------------------------------------*)
					1..2 : (* Read Coil Status / Read Input Status *)
						count := 9; (* erstes Datenbyte *)
						coils := BYTE#0;
						mask := BYTE#1;
						FOR i := 1 TO points DO
							IF mask = BYTE#0 THEN
								mask := BYTE#1;
								S_BUF.BUFFER[count] := coils;
								coils := BYTE#0;
								count := count + 1;
							END_IF;
							IF (DATA[adr1] AND SHL(WORD#1,bit_pos)) > WORD#0 THEN
								coils := coils OR mask;
							END_IF;
	
							bit_Pos := bit_Pos + 1;
							IF bit_pos > 15 THEN
								ADR1 := ADR1 + 1;
								bit_pos := 0;
							END_IF;
	
							mask := SHL(mask,1);
						END_FOR;
						S_BUF.BUFFER[Count] := coils;
	
						S_BUF.BUFFER[8] := INT_TO_BYTE(count - 8); (* Bytecount *)
						S_BUF.SIZE := INT_TO_UINT(count + 1);
	
					(*--------------------------------------------------*)
					3..4 : (* Read Holding Registers / Read Input Registers *)
						idx1 := 07;
						count := adr1 + points - 1;
						FOR i := adr1 TO count DO
							idx1 := idx1 + 2;
							idx2 := idx1 + 1; (* zweiter index für pcworx notwendig ! *)
							w_tmp := DATA[i];
							S_BUF.BUFFER[idx1] := WORD_TO_BYTE(SHR(w_tmp,8));
							S_BUF.BUFFER[idx2] := WORD_TO_BYTE(w_tmp);
						END_FOR;
						S_BUF.BUFFER[8] := SHL(INT_TO_BYTE(points),1); (* Anzahl Register in Bytes *)
						S_BUF.SIZE := INT_TO_UINT(idx2 + 1);
					(*--------------------------------------------------*)
					5 : (* Force Single Coil *)
						DATA[adr1]:=OSCAT_BASIC.BIT_LOAD_W(DATA[adr1],R_BUF.BUFFER[10] > BYTE#0,bit_pos);
						S_BUF.SIZE := UINT#12;
					(*--------------------------------------------------*)
					6 : (* Preset Single Register *)
						DATA[adr1] := OSCAT_BASIC.WORD_OF_BYTE(R_BUF.BUFFER[10],R_BUF.BUFFER[11]);
						S_BUF.SIZE := UINT#12;
					(*--------------------------------------------------*)
					15 : (* Force Multible Coils *)
						mask := BYTE#1;
						idx1 := 13;
						FOR i := 1 TO points DO
							DATA[adr1]:=OSCAT_BASIC.BIT_LOAD_W(DATA[adr1],(R_BUF.BUFFER[idx1] AND mask) > BYTE#0,bit_pos);
							bit_pos := bit_pos + 1;
							IF bit_pos > 15 THEN
								adr1:= adr1 + 1;
								bit_pos := 0;
							END_IF;
							mask := ROL(mask,1);
							IF mask = BYTE#1 THEN
								idx1 := idx1 +1;
							END_IF;
						END_FOR;
						S_BUF.SIZE := UINT#12;
					(*--------------------------------------------------*)
					16 : (* Preset Multiple Registers	*)
						idx1 := 11;
						count := adr1 + points - 1;
						FOR i := adr1 TO Count DO
							idx1 := idx1 + 2;
	 						idx2 := idx1 + 1;
							Data[i] := OSCAT_BASIC.WORD_OF_BYTE(R_BUF.BUFFER[idx1],R_BUF.BUFFER[idx2]);
						END_FOR;
						S_BUF.SIZE := UINT#12;
					(*--------------------------------------------------*)
					22 : (* Mask Write Register *)
						w_tmp := OSCAT_BASIC.WORD_OF_BYTE(R_BUF.BUFFER[10],R_BUF.BUFFER[11]); (* and mask *)
						DATA[adr1] := (DATA[adr1] AND w_tmp) OR (OSCAT_BASIC.WORD_OF_BYTE(R_BUF.BUFFER[12],R_BUF.BUFFER[13]) AND (NOT w_tmp));
						S_BUF.SIZE := UINT#14;
					(*--------------------------------------------------*)
					23 : (* Read / Write Registers	*)
						(*--- Write-Register -----------------------------------*)
						adr2 := WORD_TO_INT(OSCAT_BASIC.WORD_OF_BYTE(R_BUF.BUFFER[12],R_BUF.BUFFER[13]));
						points2 := WORD_TO_INT(OSCAT_BASIC.WORD_OF_BYTE(R_BUF.BUFFER[14],R_BUF.BUFFER[15]));
	
						(* Virtual Address Write Register *)
						MB_VMAP(VMAP:=VMAP,FC:=16,V_ADR:=adr2,V_CNT:=points2,SIZE:=DATA_SIZE);
						adr2:=MB_VMAP.P_ADR;
						ERROR:=BYTE_TO_DWORD(MB_VMAP.ERROR);
	
						IF ERROR = DWORD#0 THEN
							idx1 := 15;
							count := adr2 + points2 - 1;
							FOR i := adr2 TO count DO
								idx1 := idx1 + 2;
	 							idx2 := idx1 + 1; (* zweiter index für pcworx notwendig ! *)
								Data[i] := OSCAT_BASIC.WORD_OF_BYTE(R_BUF.BUFFER[idx1],R_BUF.BUFFER[idx2]);
							END_FOR;
	
							(*--- Read-Register -----------------------------------*)
							idx1 := 07;
							count := adr1 + points - 1;
							FOR i := adr1 TO count DO
								idx1 := idx1 + 2;
								idx2 := idx1 + 1; (* zweiter index für pcworx notwendig ! *)
								w_tmp := DATA[i];
								S_BUF.BUFFER[idx1] := WORD_TO_BYTE(SHR(w_tmp,8));
								S_BUF.BUFFER[idx2] := WORD_TO_BYTE(w_tmp);
							END_FOR;
							S_BUF.BUFFER[8] := SHL(INT_TO_BYTE(points),1); (* Anzahl Register in Bytes *)
							S_BUF.SIZE := INT_TO_UINT(idx2 + 1);
	
						END_IF;
	
					(*--------------------------------------------------*)
					ELSE
						ERROR := DWORD#01; (* ILLEGAL FUNCTION *)
					END_CASE;
				END_IF;
			END_IF;
	
			IF ERROR > DWORD#0 THEN
				S_BUF.BUFFER[7] := S_BUF.BUFFER[7] OR BYTE#2#1000_0000; (* Fehlerbit setzen *)
				S_BUF.BUFFER[8] := DWORD_TO_BYTE(ERROR);
				S_BUF.SIZE := UINT#9;
			END_IF;
	
			S_BUF.BUFFER[4] := BYTE#0; (* high Byte *)
			S_BUF.BUFFER[5] := UINT_TO_BYTE(S_BUF.SIZE - UINT#6); (* Längenfeld eintragen - nur low byte *)
	
		END_IF;
	ELSE
		ERROR := IP_C.ERROR;
	END_IF;

	t(IN:= ip_error, PT:=T#5s);
	IF t.Q THEN
		IP_C.TIME_RESET := TRUE; (* Error Reset *)
	END_IF;

	R_BUF.SIZE := UINT#0; (* Empfangsdaten zerstören *)

	IF ENABLE = FALSE THEN
	    ip_state := BYTE#4; (* Abmelden *)
		state := 00;
	END_IF;
END_CASE;

(* IP_FIFO *)
IP_FIFO(FIFO:=IP_C.FIFO,STATE:=ip_state,ID:=ip_id);

(* revision history
ks	05. jan. 2009	rev 1.0
	original version

ks	28. jan. 2009	rev 1.1
	network_buffer_short verwendet  

ks	20. oct. 2009	rev 1.2
	change lokal-var adr to adr1,Networkbuffer und Buffer-funktionen auf Basis 0

ks	17. may. 2011	rev 1.3
	automatischer re-connect
*)

END_FUNCTION_BLOCK

// POUs/DEMO/MB_SERVER_DEMO
PROGRAM MB_SERVER_DEMO
VAR
	IP_CONTROL2_1: IP_CONTROL2;
	MB_SERVER_1: MB_SERVER;
	IP_C: IP_C;
	S_BUF: NETWORK_BUFFER_SHORT;
	R_BUF: NETWORK_BUFFER_SHORT;
	DATA: ARRAY [0..255] OF WORD;
	VMAP: ARRAY [1..10] OF VMAP_DATA;
	error: DWORD;
END_VAR

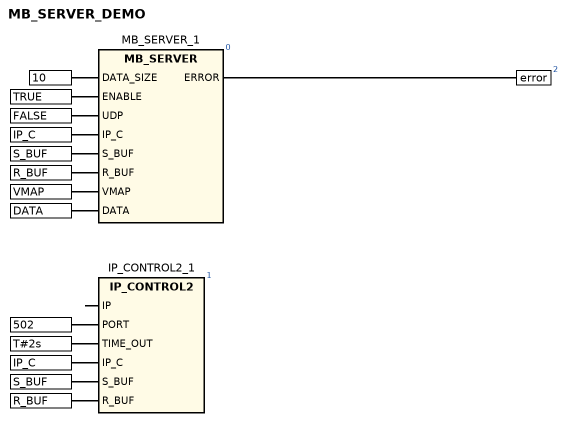
MB_SERVER_1(
    DATA_SIZE := 10,
    ENABLE := TRUE,
    UDP := FALSE,
    IP_C := IP_C,
    S_BUF := S_BUF,
    R_BUF := R_BUF,
    VMAP := VMAP,
    DATA := DATA); // MB_SERVER
IP_CONTROL2_1(PORT := 502, TIME_OUT := T#2s, IP_C := IP_C, S_BUF := S_BUF, R_BUF := R_BUF); // IP_CONTROL2
error := MB_SERVER_1.ERROR;

END_PROGRAM

// POUs/DEMO/MD5_CRAM_AUTH_DEMO
PROGRAM MD5_CRAM_AUTH_DEMO
VAR
	run: BOOL := TRUE;
	timestamp : STRING(64) := 'PDQwMzYuMTA3NjMyNDM4MUBndWlsZGVuc3Rlcm4uemVpdGZvcm0uZGU+';
	password : STRING := 'geheimes_passwort';
	username : STRING := 'benutzer@zeitform.de';
	auth_key : STRING(OSCAT_BASIC.STRING_LENGTH);
	MD5_CRAM_AUTH: MD5_CRAM_AUTH;
END_VAR

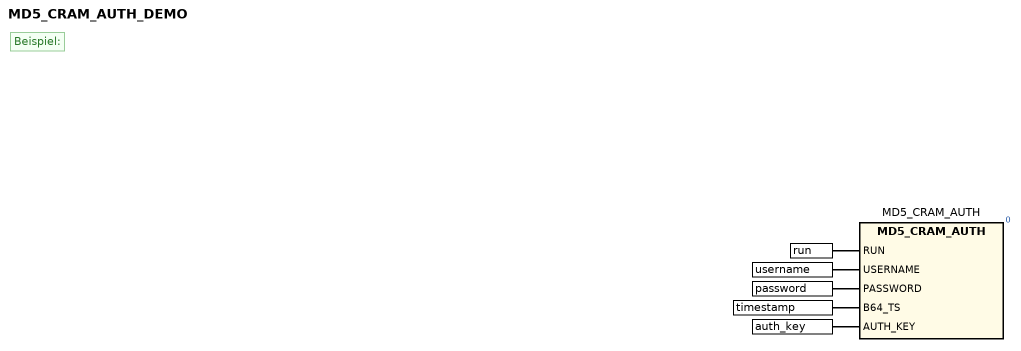
// Beispiel:
MD5_CRAM_AUTH(
    RUN := run,
    USERNAME := username,
    PASSWORD := password,
    B64_TS := timestamp,
    AUTH_KEY := auth_key);

END_PROGRAM

// POUs/CONVERT/MD5_STR
FUNCTION_BLOCK MD5_STR
VAR_INPUT
	RUN: BOOL;
END_VAR
VAR_OUTPUT
	DONE: BOOL;
END_VAR
VAR_IN_OUT
	STR: STRING(OSCAT_BASIC.STRING_LENGTH);
	MD5 : ARRAY [0..15] OF BYTE;
END_VAR
VAR
	run_last: BOOL;
	MD5_STREAM : MD5_STREAM;
	buf : ARRAY [0..63] OF BYTE;
	mode : INT;
	size : UDINT;
	pos : UDINT;
END_VAR

(*
version 1.0	06. dec. 2009
programmer 	ks
tested BY	ks

MD5_STR berechnet den MD5 Hash eines Strings
*)

CASE mode OF
0:	(* Wait für Start *)
	IF RUN AND NOT run_last THEN
		DONE := FALSE;
		mode := 1; (* Initialisierung *)
		size := LEN(STR);
	END_IF;

2:	(* Data copy and Calc *)
	IF size > 0 THEN
		OSCAT_BASIC._STRING_TO_BUFFER(STR:=MID(STR, UDINT_TO_INT(SIZE), UDINT_TO_INT(POS) + 1), POS:=0, PT:=ADR(buf), SIZE:=SIZEOF(buf));
	END_IF;

3:	DONE := TRUE;
	mode := 0; (* Stop *)

END_CASE;

IF mode > 0 THEN
	MD5_STREAM(SIZE:=size, MODE:=mode, BUF:=buf, MD5:=MD5, POS=>pos);
END_IF;

run_last := RUN;

(* revision history

ks	6. dec. 2009 rev 1.0
	original version

*)

END_FUNCTION_BLOCK

// POUs/WEATHER/MOON_PHASE
FUNCTION_BLOCK MOON_PHASE
VAR_INPUT
	XDT : DT;
	SCALE : BYTE := 12;
	UPDATE : TIME := T#1h;
END_VAR
VAR_OUTPUT
	PHASE : BYTE;
END_VAR
VAR
	x : UDINT;
	last_dt : DT;
END_VAR

(*
version 1.0		15. may. 2011
programmer		ks
tested by			ks

MOON_PHASE berechnet die aktuelle Mondphase
*)

IF XDT - last_dt > UPDATE THEN
	x := (DT_TO_UDINT(XDT) - 603240) MOD 2551392;
	PHASE := UDINT_TO_BYTE(SCALE * x / 2551392) ;
	last_dt := XDT;
END_IF;

(* revision history
ks	15.may. 2011	rev 1.0
	original version

*)

END_FUNCTION_BLOCK

// POUs/NET_VAR/NET_VAR_BOOL8
FUNCTION_BLOCK NET_VAR_BOOL8
VAR_IN_OUT
	X : NET_VAR_DATA;
END_VAR
VAR_INPUT
	IN1 : BOOL;
	IN2 : BOOL;
	IN3 : BOOL;
	IN4 : BOOL;
	IN5 : BOOL;
	IN6 : BOOL;
	IN7 : BOOL;
	IN8 : BOOL;
END_VAR
VAR_OUTPUT
	OUT1 : BOOL;
	OUT2 : BOOL;
	OUT3 : BOOL;
	OUT4 : BOOL;
	OUT5 : BOOL;
	OUT6 : BOOL;
	OUT7 : BOOL;
	OUT8 : BOOL;
	ID : BYTE;
END_VAR
VAR
	init : BOOL;
	index : INT;
	index2 : INT;
	BYTE_TO_BITS : OSCAT_BASIC.BYTE_TO_BITS;
END_VAR

(*
version 1.0		15. may. 2011
programmer		ks
tested by			ks

NET_VAR_BOOL8 überträgt bidirektional 8 boolsche Werte vom Master zum Client
*)

IF NOT init THEN
	init := TRUE;
	X.ID_MAX := X.ID_MAX + USINT#1;
	ID := USINT_TO_BYTE(X.ID_MAX);
END_IF;

IF X.STATE > BYTE#0 AND X.ERROR_ID = BYTE#0 THEN
	index := X.index; (* PCWORX Workaround *)
	IF INT_TO_UINT(index + 3) > X.BUF_SIZE THEN
		X.ERROR_ID := ID;
	ELSE
		IF X.STATE = BYTE#1 THEN (* Daten schreiben *)
			X.S_BUF.BUFFER[index] := ID; (* ID *)
			index := index + 1;
			X.S_BUF.BUFFER[index] := BYTE#4; (* TYPE BOOL8 *)
			index := index + 1;
			X.S_BUF.BUFFER[index] := OSCAT_BASIC.BYTE_OF_BIT(IN1,IN2,IN3,IN4,IN5,IN6,IN7,IN8);
			index := index + 1;

		ELSIF X.STATE = BYTE#2 THEN (* Daten lesen *)
			index2 := index + 1; (* PCWORX Workaround *)
			IF X.R_BUF.BUFFER[index] <> ID OR X.R_BUF.BUFFER[index2] <> BYTE#4 THEN
				X.ERROR_ID := ID;
			ELSE
				index := index + 2;
				BYTE_TO_BITS(IN:=X.R_BUF.BUFFER[index]);
				OUT1 := BYTE_TO_BITS.B0;
				OUT2 := BYTE_TO_BITS.B1;
				OUT3 := BYTE_TO_BITS.B2;
				OUT4 := BYTE_TO_BITS.B3;
				OUT5 := BYTE_TO_BITS.B4;
				OUT6 := BYTE_TO_BITS.B5;
				OUT7 := BYTE_TO_BITS.B6;
				OUT8 := BYTE_TO_BITS.B7;
				index := index + 1;
			END_IF;
		END_IF;
		X.index := index;
	END_IF;
END_IF;

(* revision history
ks	15.may. 2011	rev 1.0
	original version

*)

END_FUNCTION_BLOCK

// POUs/NET_VAR/NET_VAR_BUFFER
FUNCTION_BLOCK NET_VAR_BUFFER
VAR_IN_OUT
	BUF_IN : ARRAY[1..64] OF BYTE;
	BUF_OUT : ARRAY[1..64] OF BYTE;
	X : NET_VAR_DATA;
END_VAR
VAR_OUTPUT
	ID : BYTE;
END_VAR
VAR
	size : INT;
	init : BOOL;
	index : INT;
	index2 : INT;
END_VAR

(*
version 1.0		15. may. 2011
programmer		ks
tested by			ks

NET_VAR_BUFFER überträgt bidirektional 64 Bytes vom Master zum Client
*)

IF NOT init THEN
	init := TRUE;
	X.ID_MAX := X.ID_MAX + USINT#1;
	ID := USINT_TO_BYTE(X.ID_MAX);
END_IF;

IF X.STATE > BYTE#0 AND X.ERROR_ID = BYTE#0 THEN
	index := X.index; (* PCWORX Workaround *)
	IF X.STATE = BYTE#1 THEN (* Daten schreiben *)
		size := SIZEOF(BUF_IN);
		IF INT_TO_UINT(index + 3 + size) > X.BUF_SIZE THEN
			X.ERROR_ID := ID;
		ELSE
			X.S_BUF.BUFFER[index] := ID; (* ID *)
			index := index + 1;
			X.S_BUF.BUFFER[index] := BYTE#20; (* TYPE BUFFER *)
			index := index + 1;
			X.S_BUF.BUFFER[index] := INT_TO_BYTE(size); (* Anzahl der Bytes *)
				index := index + 1;
			FOR index2 := 1 TO size DO
				X.S_BUF.BUFFER[index] := BUF_IN[index2];
				index := index + 1;
			END_FOR;
		END_IF;
	ELSIF X.STATE = BYTE#2 THEN (* Daten lesen *)
		index2 := index + 1; (* PCWORX Workaround *)
		IF X.R_BUF.BUFFER[index] <> ID OR X.R_BUF.BUFFER[index2] <> BYTE#20 THEN
			X.ERROR_ID := ID;
		ELSE
			index := index + 2;
			size := BYTE_TO_INT(X.R_BUF.BUFFER[index]);
			index := index + 1;
			FOR index2 := 1 TO size DO
				BUF_OUT[index2] := X.R_BUF.BUFFER[index];
				index := index + 1;
			END_FOR;
		END_IF;
	END_IF;
	X.index := index;
END_IF;

(* revision history
ks	15.may. 2011	rev 1.0
	original version

*)

END_FUNCTION_BLOCK

// POUs/NET_VAR/NET_VAR_CONTROL
FUNCTION_BLOCK NET_VAR_CONTROL
VAR_INPUT
	ACTIVATE : BOOL;
	MASTER : BOOL;
	UDP : BOOL;
	REMOTE_IP4 : DWORD;
	REMOTE_PORT : WORD := 10000;
	SCAN_TIME : TIME := T#1s;
	WATCHDOG : TIME := T#2s;
END_VAR
VAR_OUTPUT
	RUN : BOOL;
	ERROR : DWORD;
END_VAR
VAR_IN_OUT
	X : NET_VAR_DATA;
END_VAR
VAR
	IPC : IP_CONTROL;
	IP_C : IP_C; (* IP_Control Verwaltungsstruktur *)
	step : INT;
	activate_last : BOOL;
	tscan : TON;
	reset : BOOL;
END_VAR

(*
version 1.0		15. may. 2011
programmer		ks
tested by			ks

NET_VAR_CONTROL überträgt Daten bidirektional vom Master zum Client
*)

(* Typ
001 = BYTE
002 = WORD
003 = DWORD
004 = BOOL (8x)
005 = REAL
006 = STRING
007 = UINT
008 = INT
009 = DINT
010 = UDINT
013 = DWORD (8x)
015 = REAL (8x)

020 = BUFFER
021 = MIX (REAL,DINT,UDINT,
*)

IF X.ERROR_ID > BYTE#0 THEN (* Schwere Fehler bei Variablenzuordnung vorhanden  !! *)
	X.STATE := BYTE#0;
	ERROR := BYTE_TO_DWORD(X.ERROR_ID);
	X.ERROR_ID := BYTE#0;
	step := 999;
END_IF;

CASE step OF

00:	IF ACTIVATE AND NOT activate_last OR reset THEN

        (*  TCP + MASTER = C_MODE 0 (TCP + ACTIVE + PORT + IP) *)
        (*  UDP + MASTER = C_MODE 1 (UDP + ACTIVE + PORT + IP) *)
        (*  TCP + SLAVE  = C_MODE 2 (TCP + PASSIV + PORT + IP) *)
        (*  UDP + SLAVE  = C_MODE 3 (UDP + PASSIV + PORT + IP) *)
	IF MASTER THEN
		IP_C.C_MODE := BYTE#0;
		step := 100;
	ELSE
		IP_C.C_MODE := BYTE#2;
		step := 200;
	END_IF;
        IF UDP THEN IP_C.C_MODE := IP_C.C_MODE OR BYTE#1; END_IF;
	  	IP_C.C_PORT := REMOTE_PORT; (* Portnummer eintragen *)
	  	IP_C.C_IP := REMOTE_IP4; (* IP eintragen *)
	  	IP_C.TIME_RESET := TRUE; (* Zeitueberwachung rücksetzen *)
	  	IP_C.C_ENABLE := TRUE; (* Verbindungsaufbau freigeben *)
	  	IP_C.R_OBSERVE := TRUE; (* Empfangsueberwachung *)
		X.S_BUF.SIZE := UINT#0;
		X.R_BUF.SIZE := UINT#0;
		X.CYCLE := UDINT#0;
		X.ERROR_ID := BYTE#0;
		reset := FALSE;
	END_IF;

(* ++++++++++++++++++++++++++++++++++++++++++++++ *)

100:IF IP_C.C_STATE > BYTE#127 THEN (* Verbindung vorhanden *)
		X.STATE := BYTE#1; (* Daten sammeln *)
		X.BUF_SIZE := SIZEOF(X.S_BUF.BUFFER);
		X.S_BUF.BUFFER[0] := UDINT_TO_BYTE(X.CYCLE);
		X.INDEX := 1;
		step := 110;
	END_IF;

110:X.STATE := BYTE#0;
	X.S_BUF.SIZE := INT_TO_UINT(X.INDEX); (* Datenlänge eintragen *)
	step := 120;

120:IF X.S_BUF.SIZE = UINT#0 AND X.R_BUF.SIZE >= UINT#1 THEN (* länge der empfangenen Daten prüfen *)
		X.STATE := BYTE#2; (* Daten ausgeben *)
		X.BUF_SIZE := X.R_BUF.SIZE;
		X.INDEX := 1;
		X.ERROR_ID := BYTE#0;
		X.CYCLE := X.CYCLE + UDINT#1;
		ERROR := DWORD#0; (* nach erfolgreichen Zyklus letzten Fehlercode löschen *)
		RUN := TRUE;
		step := 130;
	END_IF;

130:X.STATE := BYTE#0;
	X.R_BUF.SIZE := UINT#0;
	IF NOT ACTIVATE THEN
		step := 999; (* Beenden *)
	ELSIF tscan.Q THEN
		step := 100;
	END_IF;

(* ++++++++++++++++++++++++++++++++++++++++++++++ *)

200:IF X.R_BUF.SIZE >= UINT#1 THEN
		X.STATE := BYTE#2; (* Daten ausgeben *)
		X.BUF_SIZE := X.R_BUF.SIZE;
		X.INDEX := 1;
		step := 210;
	END_IF;

210:X.STATE := BYTE#1; (* Daten sammeln *)
	X.BUF_SIZE := SIZEOF(X.R_BUF.BUFFER);;
	X.S_BUF.BUFFER[0] := X.R_BUF.BUFFER[0]; (* Cycle übernehmen *)
	X.INDEX := 1;
	X.R_BUF.SIZE := UINT#0;
	step := 220;

220:X.STATE := BYTE#0;
	X.S_BUF.SIZE := INT_TO_UINT(X.INDEX); (* Datenlänge eintragen *)
	step := 230;

230:IF X.S_BUF.SIZE = UINT#0 THEN
		ERROR := DWORD#0; (* nach erfolgreichen Zyklus letzten Fehlercode löschen *)
		RUN := TRUE;
		IF NOT ACTIVATE THEN
			step := 999; (* Beenden *)
		ELSE
			step := 200;
		END_IF;
	END_IF;

999:IP_C.C_ENABLE := FALSE; (* Beenden *)
	RUN := FALSE;
	step := 0;

END_CASE;

(* ++++++++++++++++++++++++++++++++++++++++++++++ *)

IPC(IP:= DWORD#0, PORT:= WORD#0 , TIME_OUT:= WATCHDOG, IP_C:= IP_C, S_BUF:= X.S_BUF, R_BUF:= X.R_BUF);

IF IP_C.ERROR > DWORD#0 THEN
	ERROR := IP_C.ERROR;
	RUN := FALSE;
	reset := TRUE;
	step := 0;
END_IF;

ACTIVATE_LAST := ACTIVATE; (* letzten Status sichern zur Flankenerkennung *)
tscan(IN:= step <> 110 ,PT:=SCAN_TIME);

(* revision history
ks	15.may. 2011	rev 1.0
	original version

*)

END_FUNCTION_BLOCK

// POUs/NET_VAR/NET_VAR_DWORD8
FUNCTION_BLOCK NET_VAR_DWORD8
VAR_IN_OUT
	X : NET_VAR_DATA;
END_VAR
VAR_INPUT
	IN1 : DWORD;
	IN2 : DWORD;
	IN3 : DWORD;
	IN4 : DWORD;
	IN5 : DWORD;
	IN6 : DWORD;
	IN7 : DWORD;
	IN8 : DWORD;
END_VAR
VAR_OUTPUT
	OUT1 : DWORD;
	OUT2 : DWORD;
	OUT3 : DWORD;
	OUT4 : DWORD;
	OUT5 : DWORD;
	OUT6 : DWORD;
	OUT7 : DWORD;
	OUT8 : DWORD;
	ID : BYTE;
END_VAR
VAR
	init : BOOL;
	i : INT;
	i2 : INT;
	index : INT;
	index2 : INT;
	ra : ARRAY[1..8] OF DWORD;
END_VAR

(*
version 1.0		15. may. 2011
programmer		ks
tested by			ks

NET_VAR_DWORD8 überträgt bidirektional acht DWORD vom Master zum Client
*)

IF NOT init THEN
	init := TRUE;
	X.ID_MAX := X.ID_MAX + USINT#1;
	ID := USINT_TO_BYTE(X.ID_MAX);
END_IF;

IF X.STATE > BYTE#0 AND X.ERROR_ID = BYTE#0 THEN
	index := X.index; (* PCWORX Workaround *)
	IF INT_TO_UINT(index + 34) > X.BUF_SIZE THEN  (* ID (1) + TYPE (1) + 8 x DWORD (4) *)
		X.ERROR_ID := ID;
	ELSE
		IF X.STATE = BYTE#1 THEN (* Daten schreiben *)
			ra[1] := IN1;
			ra[2] := IN2;
			ra[3] := IN3;
			ra[4] := IN4;
			ra[5] := IN5;
			ra[6] := IN6;
			ra[7] := IN7;
			ra[8] := IN8;
			X.S_BUF.BUFFER[index] := ID; (* ID *)
			index := index + 1;
			X.S_BUF.BUFFER[index] := BYTE#13; (* TYPE DWORD8 *)
			index := index + 1;
			FOR i2 := 1 TO 8 DO;
				FOR i := 1 TO 4 DO;
					X.S_BUF.BUFFER[index] := DWORD_TO_BYTE(ra[i2]);
					ra[i2] := ROR(ra[i2],8);
					index := index + 1;
				END_FOR;
			END_FOR;

		ELSIF X.STATE = BYTE#2 THEN (* Daten lesen *)
			index2 := index + 1; (* PCWORX Workaround *)
			IF X.R_BUF.BUFFER[index] <> ID OR X.R_BUF.BUFFER[index2] <> BYTE#13 THEN (* TYPE DWORD8 *)
				X.ERROR_ID := ID;
			ELSE
				index := index + 2;
				FOR i2 := 1 TO 8 DO;
					ra[i2] := DWORD#0;
					FOR i := 1 TO 4 DO;
						ra[i2] := ra[i2] OR BYTE_TO_DWORD(X.R_BUF.BUFFER[index]);
						ra[i2] := ROR(ra[i2],8);
						index := index + 1;
					END_FOR;
				END_FOR;
				OUT1 := ra[1];
				OUT2 := ra[2];
				OUT3 := ra[3];
				OUT4 := ra[4];
				OUT5 := ra[5];
				OUT6 := ra[6];
				OUT7 := ra[7];
				OUT8 := ra[8];
			END_IF;
		END_IF;
		X.index := index;
	END_IF;
END_IF;

(* revision history
ks	15.may. 2011	rev 1.0
	original version

*)

END_FUNCTION_BLOCK

// POUs/DEMO/NET_VAR_MASTER_DEMO
PROGRAM NET_VAR_MASTER_DEMO
VAR
	NET_VAR_CONTROL_1: NET_VAR_CONTROL;
	activate: BOOL := TRUE;
	run: BOOL;
	udp: BOOL := TRUE;
	master: BOOL := TRUE;
	remote_port: WORD := 10000;
	scan_time: TIME := T#1s;
	watchdog: TIME := T#2s;
	error: DWORD;
	x: NET_VAR_DATA;

	NET_VAR_BOOL8_1: NET_VAR_BOOL8;
	id_b8: BYTE;
	in_b1: BOOL;
	in_b2: BOOL;
	in_b3: BOOL;
	in_b4: BOOL;
	in_b5: BOOL;
	in_b6: BOOL;
	in_b7: BOOL;
	in_b8: BOOL;
	out_b1: BOOL;
	out_b2: BOOL;
	out_b3: BOOL;
	out_b4: BOOL;
	out_b5: BOOL;
	out_b6: BOOL;
	out_b7: BOOL;
	out_b8: BOOL;

	NET_VAR_STRING_1: NET_VAR_STRING;
	in_s1: STRING(OSCAT_BASIC.STRING_LENGTH);
	out_s1: STRING(OSCAT_BASIC.STRING_LENGTH);
	id_s: BYTE;

	NET_VAR_BUFFER_1: NET_VAR_BUFFER;
	id_bu: BYTE;
	BUF_IN : ARRAY [1..64] OF BYTE;
	BUF_OUT : ARRAY [1..64] OF BYTE;

	id_dw: BYTE;
	NET_VAR_DWORD8_1: NET_VAR_DWORD8;
	in_dw1 : DWORD;
	in_dw2 : DWORD;
	in_dw3 : DWORD;
	in_dw4 : DWORD;
	in_dw5 : DWORD;
	in_dw6 : DWORD;
	in_dw7 : DWORD;
	in_dw8 : DWORD;
	out_dw1 : DWORD;
	out_dw2 : DWORD;
	out_dw3 : DWORD;
	out_dw4 : DWORD;
	out_dw5 : DWORD;
	out_dw6 : DWORD;
	out_dw7 : DWORD;
	out_dw8 : DWORD;

	NET_VAR_REAL8_1: NET_VAR_REAL8;
	in_r1 : REAL;
	in_r2 : REAL;
	in_r3 : REAL;
	in_r4 : REAL;
	in_r5 : REAL;
	in_r6 : REAL;
	in_r7 : REAL;
	in_r8 : REAL;
	out_r1 : REAL;
	out_r2 : REAL;
	out_r3 : REAL;
	out_r4 : REAL;
	out_r5 : REAL;
	out_r6 : REAL;
	out_r7 : REAL;
	out_r8 : REAL;
	id_r: BYTE;

	NET_VAR_X8_1: NET_VAR_X8;
	in_x_re1 : REAL;
	in_x_re2 : REAL;
	in_x_di1 : DINT;
	in_x_di2 : DINT;
	in_x_ud1 : UDINT;
	in_x_ud2 : UDINT;
	in_x_dw1 : DWORD;
	in_x_dw2 : DWORD;
	out_x_re1 : REAL;
	out_x_re2 : REAL;
	out_x_di1 : DINT;
	out_x_di2 : DINT;
	out_x_ud1 : UDINT;
	out_x_ud2 : UDINT;
	out_x_dw1 : DWORD;
	out_x_dw2 : DWORD;
	id_x8: BYTE;
END_VAR
VAR // added by the converter: edge detectors and wires of the graphical bodies
    _w1 : ANY;
END_VAR

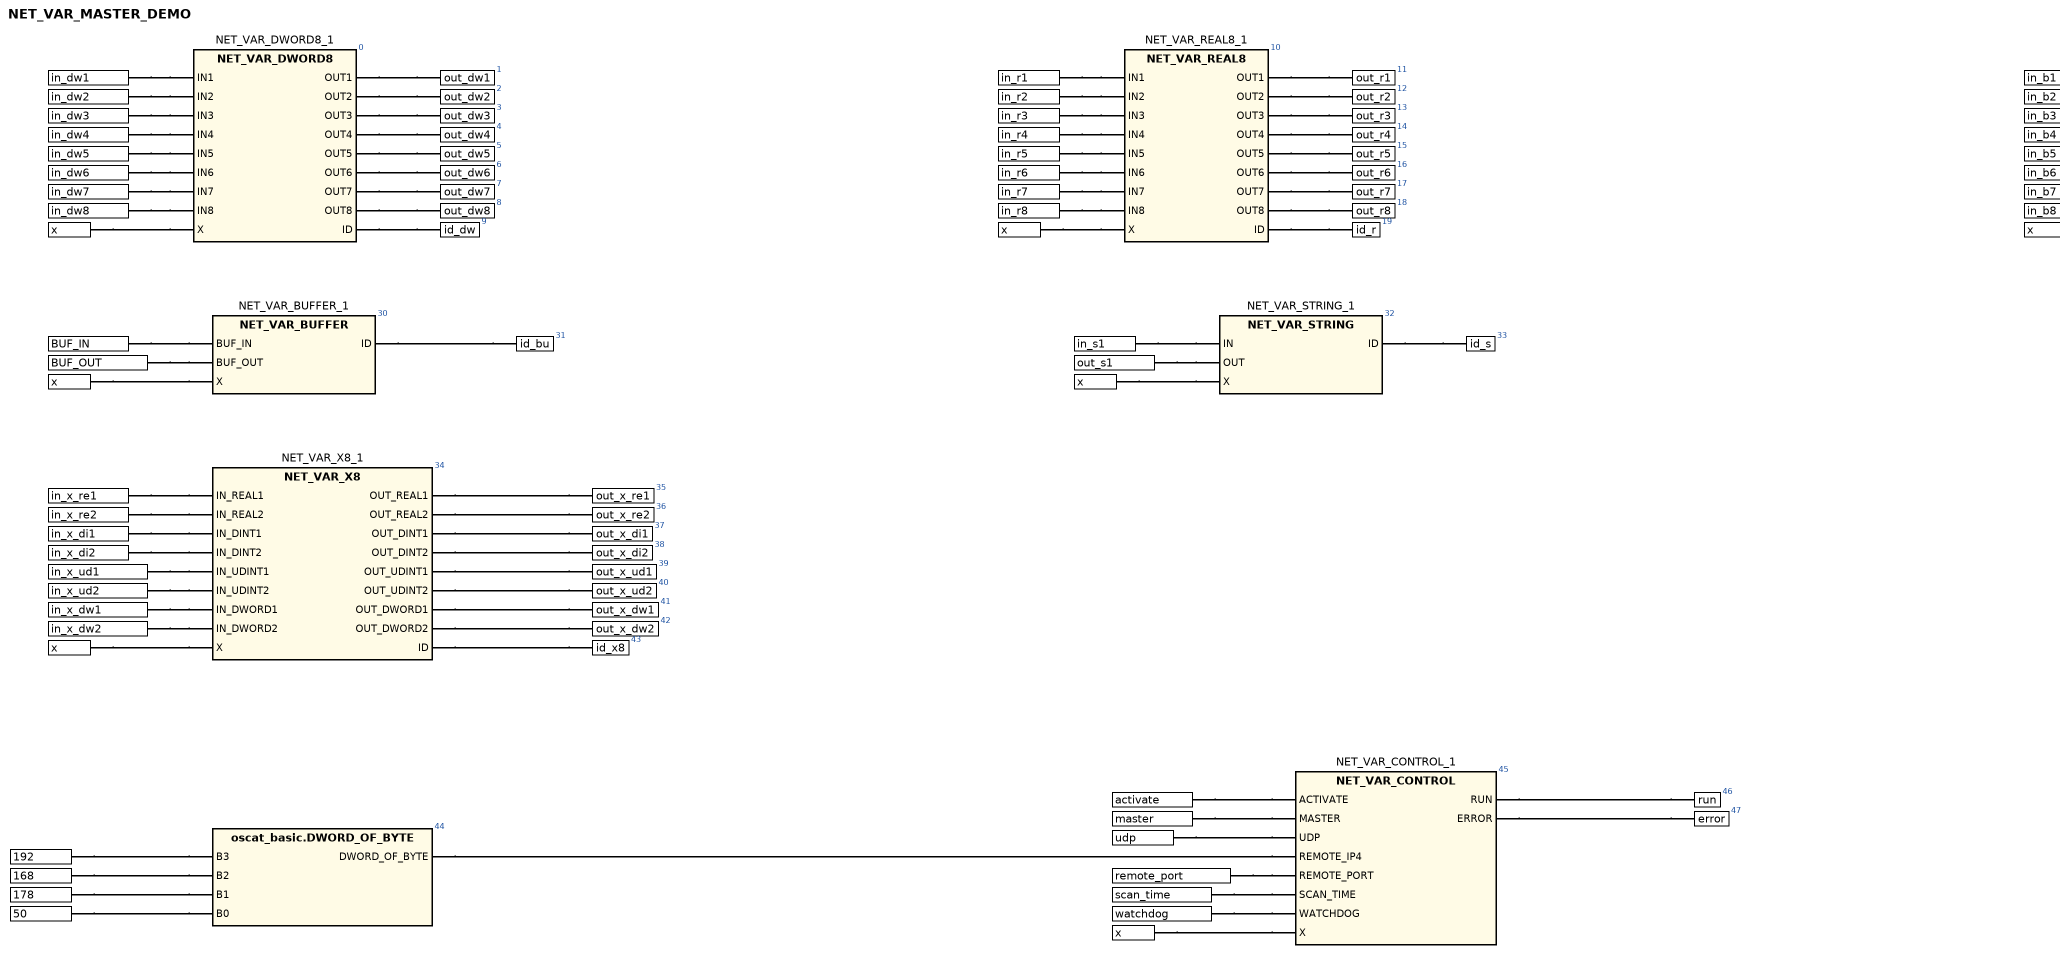
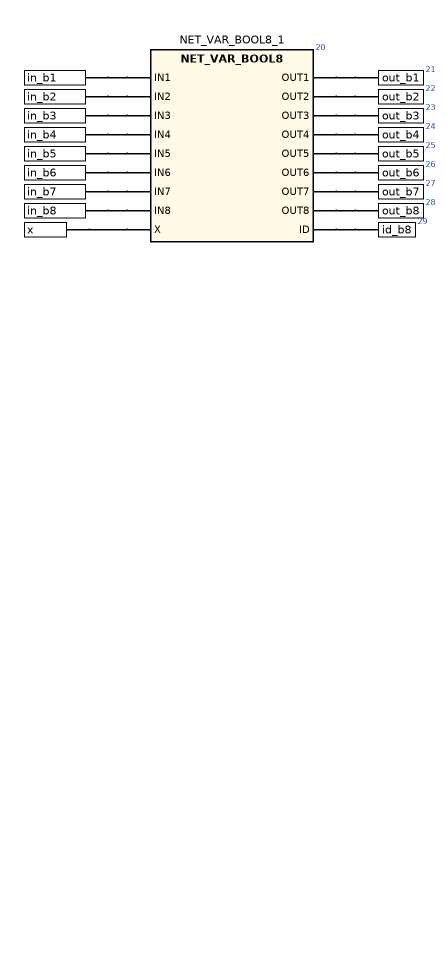
NET_VAR_DWORD8_1(
    IN1 := in_dw1,
    IN2 := in_dw2,
    IN3 := in_dw3,
    IN4 := in_dw4,
    IN5 := in_dw5,
    IN6 := in_dw6,
    IN7 := in_dw7,
    IN8 := in_dw8,
    X := x); // NET_VAR_DWORD8
out_dw1 := NET_VAR_DWORD8_1.OUT1;
out_dw2 := NET_VAR_DWORD8_1.OUT2;
out_dw3 := NET_VAR_DWORD8_1.OUT3;
out_dw4 := NET_VAR_DWORD8_1.OUT4;
out_dw5 := NET_VAR_DWORD8_1.OUT5;
out_dw6 := NET_VAR_DWORD8_1.OUT6;
out_dw7 := NET_VAR_DWORD8_1.OUT7;
out_dw8 := NET_VAR_DWORD8_1.OUT8;
id_dw := NET_VAR_DWORD8_1.ID;
NET_VAR_REAL8_1(
    IN1 := in_r1,
    IN2 := in_r2,
    IN3 := in_r3,
    IN4 := in_r4,
    IN5 := in_r5,
    IN6 := in_r6,
    IN7 := in_r7,
    IN8 := in_r8,
    X := x); // NET_VAR_REAL8
out_r1 := NET_VAR_REAL8_1.OUT1;
out_r2 := NET_VAR_REAL8_1.OUT2;
out_r3 := NET_VAR_REAL8_1.OUT3;
out_r4 := NET_VAR_REAL8_1.OUT4;
out_r5 := NET_VAR_REAL8_1.OUT5;
out_r6 := NET_VAR_REAL8_1.OUT6;
out_r7 := NET_VAR_REAL8_1.OUT7;
out_r8 := NET_VAR_REAL8_1.OUT8;
id_r := NET_VAR_REAL8_1.ID;
NET_VAR_BOOL8_1(
    IN1 := in_b1,
    IN2 := in_b2,
    IN3 := in_b3,
    IN4 := in_b4,
    IN5 := in_b5,
    IN6 := in_b6,
    IN7 := in_b7,
    IN8 := in_b8,
    X := x); // NET_VAR_BOOL8
out_b1 := NET_VAR_BOOL8_1.OUT1;
out_b2 := NET_VAR_BOOL8_1.OUT2;
out_b3 := NET_VAR_BOOL8_1.OUT3;
out_b4 := NET_VAR_BOOL8_1.OUT4;
out_b5 := NET_VAR_BOOL8_1.OUT5;
out_b6 := NET_VAR_BOOL8_1.OUT6;
out_b7 := NET_VAR_BOOL8_1.OUT7;
out_b8 := NET_VAR_BOOL8_1.OUT8;
id_b8 := NET_VAR_BOOL8_1.ID;
NET_VAR_BUFFER_1(BUF_IN := BUF_IN, BUF_OUT := BUF_OUT, X := x); // NET_VAR_BUFFER
id_bu := NET_VAR_BUFFER_1.ID;
NET_VAR_STRING_1(IN := in_s1, OUT := out_s1, X := x); // NET_VAR_STRING
id_s := NET_VAR_STRING_1.ID;
NET_VAR_X8_1(
    IN_REAL1 := in_x_re1,
    IN_REAL2 := in_x_re2,
    IN_DINT1 := in_x_di1,
    IN_DINT2 := in_x_di2,
    IN_UDINT1 := in_x_ud1,
    IN_UDINT2 := in_x_ud2,
    IN_DWORD1 := in_x_dw1,
    IN_DWORD2 := in_x_dw2,
    X := x); // NET_VAR_X8
out_x_re1 := NET_VAR_X8_1.OUT_REAL1;
out_x_re2 := NET_VAR_X8_1.OUT_REAL2;
out_x_di1 := NET_VAR_X8_1.OUT_DINT1;
out_x_di2 := NET_VAR_X8_1.OUT_DINT2;
out_x_ud1 := NET_VAR_X8_1.OUT_UDINT1;
out_x_ud2 := NET_VAR_X8_1.OUT_UDINT2;
out_x_dw1 := NET_VAR_X8_1.OUT_DWORD1;
out_x_dw2 := NET_VAR_X8_1.OUT_DWORD2;
id_x8 := NET_VAR_X8_1.ID;
_w1 := oscat_basic.DWORD_OF_BYTE(B3 := 192, B2 := 168, B1 := 178, B0 := 50);
NET_VAR_CONTROL_1(
    ACTIVATE := activate,
    MASTER := master,
    UDP := udp,
    REMOTE_IP4 := _w1,
    REMOTE_PORT := remote_port,
    SCAN_TIME := scan_time,
    WATCHDOG := watchdog,
    X := x); // NET_VAR_CONTROL
run := NET_VAR_CONTROL_1.RUN;
error := NET_VAR_CONTROL_1.ERROR;

END_PROGRAM

// POUs/NET_VAR/NET_VAR_REAL8
FUNCTION_BLOCK NET_VAR_REAL8
VAR_IN_OUT
	X : NET_VAR_DATA;
END_VAR
VAR_INPUT
	IN1 : REAL;
	IN2 : REAL;
	IN3 : REAL;
	IN4 : REAL;
	IN5 : REAL;
	IN6 : REAL;
	IN7 : REAL;
	IN8 : REAL;
END_VAR
VAR_OUTPUT
	OUT1 : REAL;
	OUT2 : REAL;
	OUT3 : REAL;
	OUT4 : REAL;
	OUT5 : REAL;
	OUT6 : REAL;
	OUT7 : REAL;
	OUT8 : REAL;
	ID : BYTE;
END_VAR
VAR
	init : BOOL;
	i : INT;
	i2 : INT;
	index : INT;
	index2 : INT;
	r_dw : DWORD;
	ra : ARRAY[1..8] OF REAL;
END_VAR

(*
version 1.0		15. may. 2011
programmer		ks
tested by			ks

NET_VAR_REAL8 überträgt bidirektional acht REAL-Werte vom Master zum Client
*)

IF NOT init THEN
	init := TRUE;
	X.ID_MAX := X.ID_MAX + USINT#1;
	ID := USINT_TO_BYTE(X.ID_MAX);
END_IF;

IF X.STATE > BYTE#0 AND X.ERROR_ID = BYTE#0 THEN
	index := X.index; (* PCWORX Workaround *)
	IF INT_TO_UINT(index + 34) > X.BUF_SIZE THEN (* ID (1) + TYPE (1) + 8 x REAL (4) *)
		X.ERROR_ID := ID;
	ELSE
		IF X.STATE = BYTE#1 THEN (* Daten schreiben *)
			ra[1] := IN1;
			ra[2] := IN2;
			ra[3] := IN3;
			ra[4] := IN4;
			ra[5] := IN5;
			ra[6] := IN6;
			ra[7] := IN7;
			ra[8] := IN8;
			X.S_BUF.BUFFER[index] := ID; (* ID *)
			index := index + 1;
			X.S_BUF.BUFFER[index] := BYTE#15; (* TYPE REAL8 *)
			index := index + 1;
			FOR i2 := 1 TO 8 DO;
				r_dw := OSCAT_BASIC.REAL_TO_DW(X:=ra[i2]);
				FOR i := 1 TO 4 DO;
					X.S_BUF.BUFFER[index] := DWORD_TO_BYTE(r_dw);
					r_dw := ROR(r_dw,8);
					index := index + 1;
				END_FOR;
			END_FOR;

		ELSIF X.STATE = BYTE#2 THEN (* Daten lesen *)
			index2 := index + 1; (* PCWORX Workaround *)
			IF X.R_BUF.BUFFER[index] <> ID OR X.R_BUF.BUFFER[index2] <> BYTE#15 THEN (* TYPE REAL8 *)
				X.ERROR_ID := ID;
			ELSE
				index := index + 2;
				FOR i2 := 1 TO 8 DO;
					r_dw := DWORD#0;
					FOR i := 1 TO 4 DO;
						r_dw := r_dw OR BYTE_TO_DWORD(X.R_BUF.BUFFER[index]);
						r_dw := ROR(r_dw,8);
						index := index + 1;
					END_FOR;
					ra[i2] := OSCAT_BASIC.DW_TO_REAL(X:=r_dw);
				END_FOR;
				OUT1 := ra[1];
				OUT2 := ra[2];
				OUT3 := ra[3];
				OUT4 := ra[4];
				OUT5 := ra[5];
				OUT6 := ra[6];
				OUT7 := ra[7];
				OUT8 := ra[8];
			END_IF;
		END_IF;
		X.index := index;
	END_IF;
END_IF;

(* revision history
ks	15.may. 2011	rev 1.0
	original version

*)

END_FUNCTION_BLOCK

// POUs/NET_VAR/NET_VAR_STRING
FUNCTION_BLOCK NET_VAR_STRING
VAR_IN_OUT
	IN : STRING(OSCAT_BASIC.STRING_LENGTH);
	OUT : STRING(OSCAT_BASIC.STRING_LENGTH);
	X : NET_VAR_DATA;
END_VAR
VAR_OUTPUT
	ID : BYTE;
END_VAR
VAR
	init : BOOL;
	len_str : INT;
	index : INT;
	index2 : INT;
END_VAR

(*
version 1.0		15. may. 2011
programmer		ks
tested by			ks

NET_VAR_STRING überträgt bidirektional einen STRING vom Master zum Client
*)

IF NOT init THEN
	init := TRUE;
	X.ID_MAX := X.ID_MAX + USINT#1;
	ID := USINT_TO_BYTE(X.ID_MAX);
END_IF;

IF X.STATE > BYTE#0 AND X.ERROR_ID = BYTE#0 THEN
	index := X.index; (* PCWORX Workaround *)
	IF X.STATE = BYTE#1 THEN (* Daten schreiben *)
		len_str := LEN(IN);
		IF INT_TO_UINT(index + 3 + len_str) > X.BUF_SIZE THEN
			X.ERROR_ID := ID;
		ELSE
			X.S_BUF.BUFFER[index] := ID; (* ID *)
			index := index + 1;
			X.S_BUF.BUFFER[index] := BYTE#6; (* TYPE REAL *)
			index := index + 1;
			X.S_BUF.BUFFER[index] := INT_TO_BYTE(len_str); (* Anzahl der Bytes *)
			index := index + 1;
			OSCAT_BASIC._STRING_TO_BUFFER(STR:=IN,POS:=index,PT:=ADR(X.S_BUF.BUFFER),SIZE:=X.BUF_SIZE);
			index := index + len_str;
		END_IF;
	ELSIF X.STATE = BYTE#2 THEN (* Daten lesen *)
		index2 := index + 1; (* PCWORX Workaround *)
		IF X.R_BUF.BUFFER[index] <> ID OR X.R_BUF.BUFFER[index2] <> BYTE#6 THEN
			X.ERROR_ID := ID;
		ELSE
			index := index + 2;
			len_str := BYTE_TO_INT(X.R_BUF.BUFFER[index]);
			index2 := index + 1;
			index := index2 + len_str;
			IF len_STR > 0 THEN
				OUT := OSCAT_BASIC.BUFFER_TO_STRING(PT:=ADR(X.R_BUF.BUFFER),SIZE:=X.BUF_SIZE,START:=INT_TO_UINT(index2),STOP:=INT_TO_UINT(index - 1));
			ELSE
				OUT := '';
			END_IF;
		END_IF;
	END_IF;
	X.index := index;
END_IF;

(* revision history
ks	15.may. 2011	rev 1.0
	original version

*)

END_FUNCTION_BLOCK

// POUs/NET_VAR/NET_VAR_X8
FUNCTION_BLOCK NET_VAR_X8
VAR_IN_OUT
	X : NET_VAR_DATA;
END_VAR
VAR_INPUT
	IN_REAL1 : REAL;
	IN_REAL2 : REAL;
	IN_DINT1 : DINT;
	IN_DINT2 : DINT;
	IN_UDINT1 : UDINT;
	IN_UDINT2 : UDINT;
	IN_DWORD1 : DWORD;
	IN_DWORD2 : DWORD;
END_VAR
VAR_OUTPUT
	OUT_REAL1 : REAL;
	OUT_REAL2: REAL;
	OUT_DINT1 : DINT;
	OUT_DINT2 : DINT;
	OUT_UDINT1 : UDINT;
	OUT_UDINT2 : UDINT;
	OUT_DWORD1 : DWORD;
	OUT_DWORD2 : DWORD;
	ID : BYTE;
END_VAR
VAR
	init : BOOL;
	i : INT;
	i2 : INT;
	index : INT;
	index2 : INT;
	ra : ARRAY[1..8] OF DWORD;
END_VAR

(*
version 1.0		15. may. 2011
programmer		ks
tested by			ks

NET_VAR_X8 überträgt bidirektional 2x REAL,2x DINT,2x UDINT,2x DWORD vom Master zum Client
*)

IF NOT init THEN
	init := TRUE;
	X.ID_MAX := X.ID_MAX + USINT#1;
	ID := USINT_TO_BYTE(X.ID_MAX);
END_IF;

IF X.STATE > BYTE#0 AND X.ERROR_ID = BYTE#0 THEN
	index := X.index; (* PCWORX Workaround *)
	IF INT_TO_UINT(index + 34) > X.BUF_SIZE THEN  (* ID (1) + TYPE (1) + 8 x DWORD (4) *)
		X.ERROR_ID := ID;
	ELSE
		IF X.STATE = BYTE#1 THEN (* Daten schreiben *)
			ra[1] := OSCAT_BASIC.REAL_TO_DW(X:=IN_REAL1);
			ra[2] := OSCAT_BASIC.REAL_TO_DW(X:=IN_REAL2);
			ra[3] := DINT_TO_DWORD(IN_DINT1);
			ra[4] := DINT_TO_DWORD(IN_DINT2);
			ra[5] := UDINT_TO_DWORD(IN_UDINT1);
			ra[6] := UDINT_TO_DWORD(IN_UDINT2);
			ra[7] := IN_DWORD1;
			ra[8] := IN_DWORD2;
			X.S_BUF.BUFFER[index] := ID; (* ID *)
			index := index + 1;
			X.S_BUF.BUFFER[index] := BYTE#21; (* TYPE X8 *)
			index := index + 1;
			FOR i2 := 1 TO 8 DO;
				FOR i := 1 TO 4 DO;
					X.S_BUF.BUFFER[index] := DWORD_TO_BYTE(ra[i2]);
					ra[i2] := ROR(ra[i2],8);
					index := index + 1;
				END_FOR;
			END_FOR;

		ELSIF X.STATE = BYTE#2 THEN (* Daten lesen *)
			index2 := index + 1; (* PCWORX Workaround *)
			IF X.R_BUF.BUFFER[index] <> ID OR X.R_BUF.BUFFER[index2] <> BYTE#21 THEN (* TYPE X8 *)
				X.ERROR_ID := ID;
			ELSE
				index := index + 2;
				FOR i2 := 1 TO 8 DO;
					ra[i2] := DWORD#0;
					FOR i := 1 TO 4 DO;
						ra[i2] := ra[i2] OR BYTE_TO_DWORD(X.R_BUF.BUFFER[index]);
						ra[i2] := ROR(ra[i2],8);
						index := index + 1;
					END_FOR;
				END_FOR;
				OUT_REAL1 := OSCAT_BASIC.DW_TO_REAL(X:=ra[1]);
				OUT_REAL2 := OSCAT_BASIC.DW_TO_REAL(X:=ra[2]);
				OUT_DINT1 := DWORD_TO_DINT(ra[3]);
				OUT_DINT2 := DWORD_TO_DINT(ra[4]);
				OUT_UDINT1 := DWORD_TO_UDINT(ra[5]);
				OUT_UDINT2 := DWORD_TO_UDINT(ra[6]);
				OUT_DWORD1 := ra[7];
				OUT_DWORD2 := ra[8];
			END_IF;
		END_IF;
		X.index := index;
	END_IF;
END_IF;

(* revision history
ks	15.may. 2011	rev 1.0
	original version

*)

END_FUNCTION_BLOCK

// POUs/DEMO/NET_VAR_SLAVE_DEMO
PROGRAM NET_VAR_SLAVE_DEMO
VAR
	NET_VAR_CONTROL_1: NET_VAR_CONTROL;
	activate: BOOL := TRUE;
	run: BOOL;
	udp: BOOL := TRUE;
	master: BOOL := FALSE;
	remote_port: WORD := 10000;
	scan_time: TIME := T#1s;
	watchdog: TIME := T#2s;
	error: DWORD;
	x: NET_VAR_DATA;

	NET_VAR_BOOL8_1: NET_VAR_BOOL8;
	id_b8: BYTE;
	in_b1: BOOL;
	in_b2: BOOL;
	in_b3: BOOL;
	in_b4: BOOL;
	in_b5: BOOL;
	in_b6: BOOL;
	in_b7: BOOL;
	in_b8: BOOL;
	out_b1: BOOL;
	out_b2: BOOL;
	out_b3: BOOL;
	out_b4: BOOL;
	out_b5: BOOL;
	out_b6: BOOL;
	out_b7: BOOL;
	out_b8: BOOL;

	NET_VAR_STRING_1: NET_VAR_STRING;
	in_s1: STRING(OSCAT_BASIC.STRING_LENGTH);
	out_s1: STRING(OSCAT_BASIC.STRING_LENGTH);
	id_s: BYTE;

	NET_VAR_BUFFER_1: NET_VAR_BUFFER;
	id_bu: BYTE;
	BUF_IN : ARRAY [1..64] OF BYTE;
	BUF_OUT : ARRAY [1..64] OF BYTE;

	id_dw: BYTE;
	NET_VAR_DWORD8_1: NET_VAR_DWORD8;
	in_dw1 : DWORD;
	in_dw2 : DWORD;
	in_dw3 : DWORD;
	in_dw4 : DWORD;
	in_dw5 : DWORD;
	in_dw6 : DWORD;
	in_dw7 : DWORD;
	in_dw8 : DWORD;
	out_dw1 : DWORD;
	out_dw2 : DWORD;
	out_dw3 : DWORD;
	out_dw4 : DWORD;
	out_dw5 : DWORD;
	out_dw6 : DWORD;
	out_dw7 : DWORD;
	out_dw8 : DWORD;

	NET_VAR_REAL8_1: NET_VAR_REAL8;
	in_r1 : REAL;
	in_r2 : REAL;
	in_r3 : REAL;
	in_r4 : REAL;
	in_r5 : REAL;
	in_r6 : REAL;
	in_r7 : REAL;
	in_r8 : REAL;
	out_r1 : REAL;
	out_r2 : REAL;
	out_r3 : REAL;
	out_r4 : REAL;
	out_r5 : REAL;
	out_r6 : REAL;
	out_r7 : REAL;
	out_r8 : REAL;
	id_r: BYTE;

	NET_VAR_X8_1: NET_VAR_X8;
	in_x_re1 : REAL;
	in_x_re2 : REAL;
	in_x_di1 : DINT;
	in_x_di2 : DINT;
	in_x_ud1 : UDINT;
	in_x_ud2 : UDINT;
	in_x_dw1 : DWORD;
	in_x_dw2 : DWORD;
	out_x_re1 : REAL;
	out_x_re2 : REAL;
	out_x_di1 : DINT;
	out_x_di2 : DINT;
	out_x_ud1 : UDINT;
	out_x_ud2 : UDINT;
	out_x_dw1 : DWORD;
	out_x_dw2 : DWORD;
	id_x8: BYTE;
END_VAR
VAR // added by the converter: edge detectors and wires of the graphical bodies
    _w1 : ANY;
END_VAR

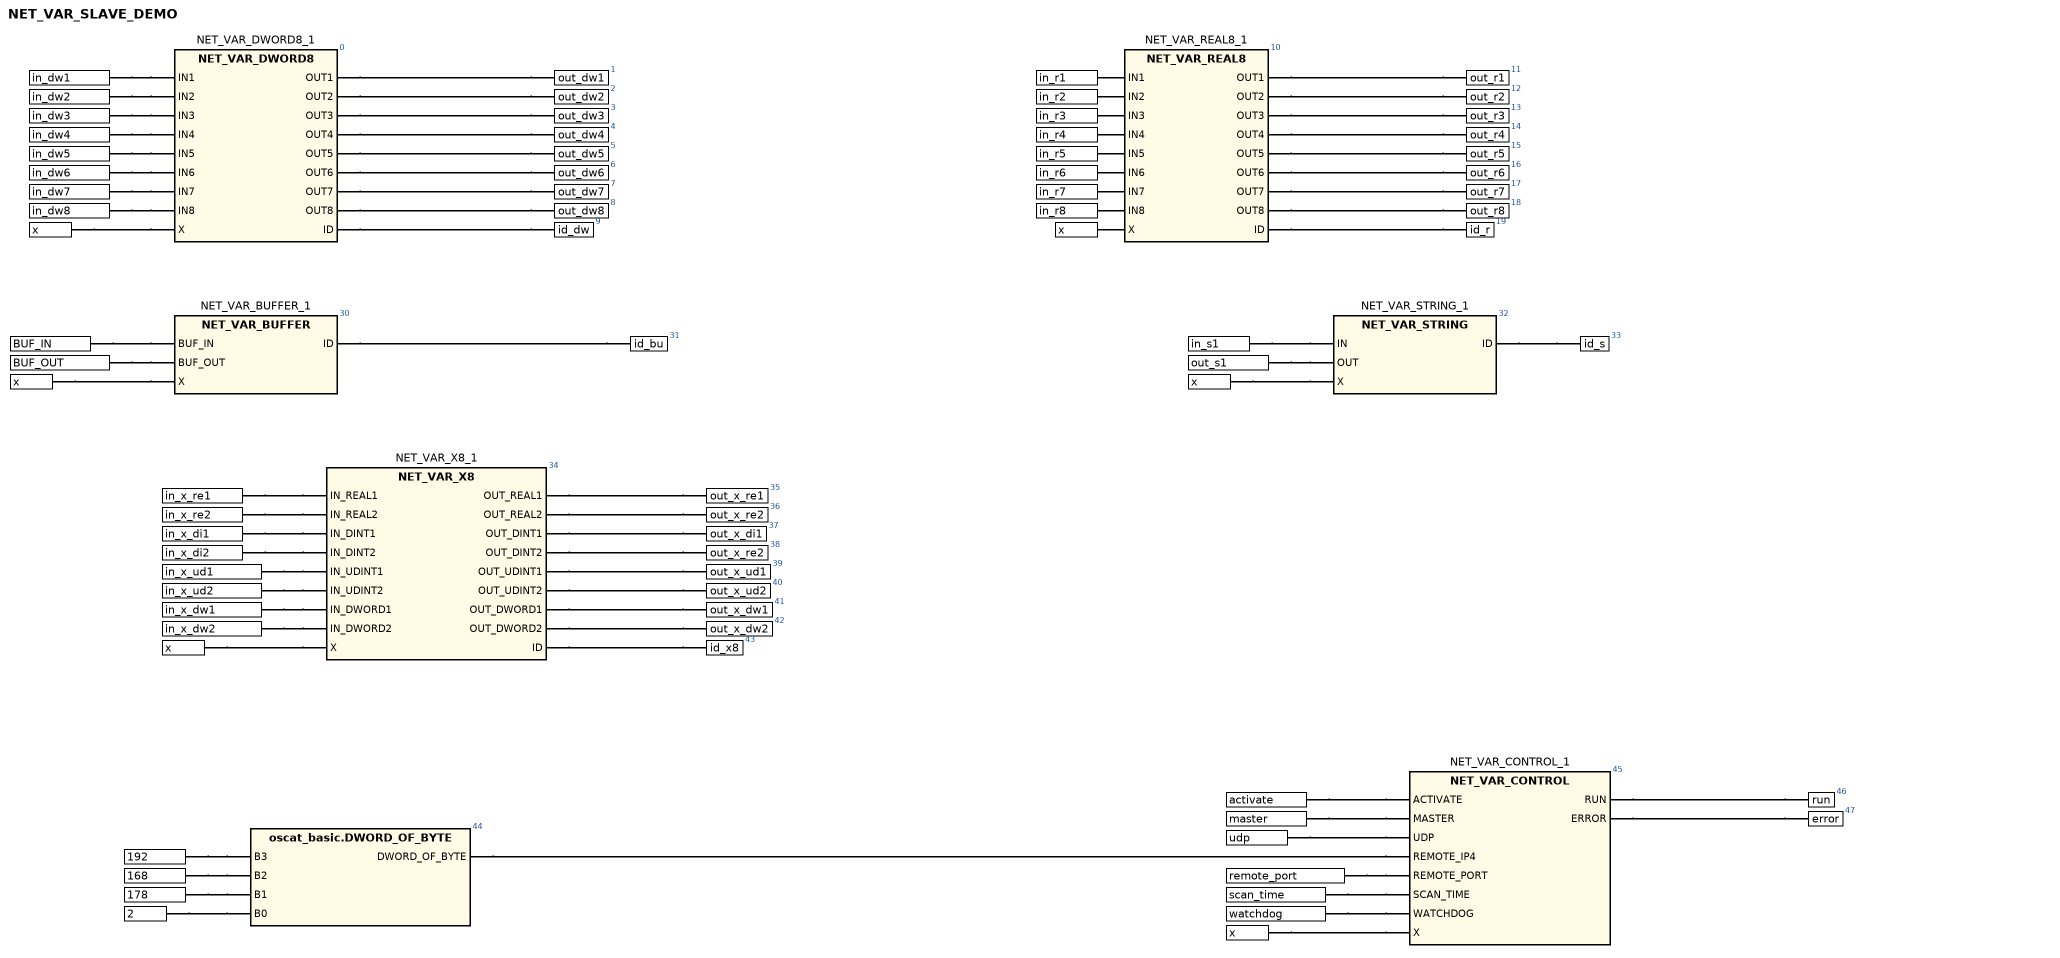
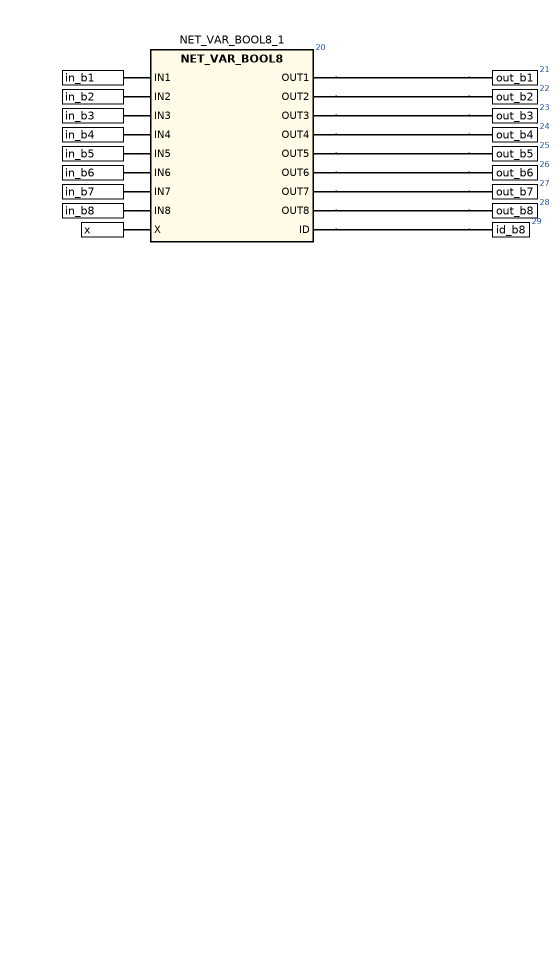
NET_VAR_DWORD8_1(
    IN1 := in_dw1,
    IN2 := in_dw2,
    IN3 := in_dw3,
    IN4 := in_dw4,
    IN5 := in_dw5,
    IN6 := in_dw6,
    IN7 := in_dw7,
    IN8 := in_dw8,
    X := x); // NET_VAR_DWORD8
out_dw1 := NET_VAR_DWORD8_1.OUT1;
out_dw2 := NET_VAR_DWORD8_1.OUT2;
out_dw3 := NET_VAR_DWORD8_1.OUT3;
out_dw4 := NET_VAR_DWORD8_1.OUT4;
out_dw5 := NET_VAR_DWORD8_1.OUT5;
out_dw6 := NET_VAR_DWORD8_1.OUT6;
out_dw7 := NET_VAR_DWORD8_1.OUT7;
out_dw8 := NET_VAR_DWORD8_1.OUT8;
id_dw := NET_VAR_DWORD8_1.ID;
NET_VAR_REAL8_1(
    IN1 := in_r1,
    IN2 := in_r2,
    IN3 := in_r3,
    IN4 := in_r4,
    IN5 := in_r5,
    IN6 := in_r6,
    IN7 := in_r7,
    IN8 := in_r8,
    X := x); // NET_VAR_REAL8
out_r1 := NET_VAR_REAL8_1.OUT1;
out_r2 := NET_VAR_REAL8_1.OUT2;
out_r3 := NET_VAR_REAL8_1.OUT3;
out_r4 := NET_VAR_REAL8_1.OUT4;
out_r5 := NET_VAR_REAL8_1.OUT5;
out_r6 := NET_VAR_REAL8_1.OUT6;
out_r7 := NET_VAR_REAL8_1.OUT7;
out_r8 := NET_VAR_REAL8_1.OUT8;
id_r := NET_VAR_REAL8_1.ID;
NET_VAR_BOOL8_1(
    IN1 := in_b1,
    IN2 := in_b2,
    IN3 := in_b3,
    IN4 := in_b4,
    IN5 := in_b5,
    IN6 := in_b6,
    IN7 := in_b7,
    IN8 := in_b8,
    X := x); // NET_VAR_BOOL8
out_b1 := NET_VAR_BOOL8_1.OUT1;
out_b2 := NET_VAR_BOOL8_1.OUT2;
out_b3 := NET_VAR_BOOL8_1.OUT3;
out_b4 := NET_VAR_BOOL8_1.OUT4;
out_b5 := NET_VAR_BOOL8_1.OUT5;
out_b6 := NET_VAR_BOOL8_1.OUT6;
out_b7 := NET_VAR_BOOL8_1.OUT7;
out_b8 := NET_VAR_BOOL8_1.OUT8;
id_b8 := NET_VAR_BOOL8_1.ID;
NET_VAR_BUFFER_1(BUF_IN := BUF_IN, BUF_OUT := BUF_OUT, X := x); // NET_VAR_BUFFER
id_bu := NET_VAR_BUFFER_1.ID;
NET_VAR_STRING_1(IN := in_s1, OUT := out_s1, X := x); // NET_VAR_STRING
id_s := NET_VAR_STRING_1.ID;
NET_VAR_X8_1(
    IN_REAL1 := in_x_re1,
    IN_REAL2 := in_x_re2,
    IN_DINT1 := in_x_di1,
    IN_DINT2 := in_x_di2,
    IN_UDINT1 := in_x_ud1,
    IN_UDINT2 := in_x_ud2,
    IN_DWORD1 := in_x_dw1,
    IN_DWORD2 := in_x_dw2,
    X := x); // NET_VAR_X8
out_x_re1 := NET_VAR_X8_1.OUT_REAL1;
out_x_re2 := NET_VAR_X8_1.OUT_REAL2;
out_x_di1 := NET_VAR_X8_1.OUT_DINT1;
out_x_re2 := NET_VAR_X8_1.OUT_DINT2;
out_x_ud1 := NET_VAR_X8_1.OUT_UDINT1;
out_x_ud2 := NET_VAR_X8_1.OUT_UDINT2;
out_x_dw1 := NET_VAR_X8_1.OUT_DWORD1;
out_x_dw2 := NET_VAR_X8_1.OUT_DWORD2;
id_x8 := NET_VAR_X8_1.ID;
_w1 := oscat_basic.DWORD_OF_BYTE(B3 := 192, B2 := 168, B1 := 178, B0 := 2);
NET_VAR_CONTROL_1(
    ACTIVATE := activate,
    MASTER := master,
    UDP := udp,
    REMOTE_IP4 := _w1,
    REMOTE_PORT := remote_port,
    SCAN_TIME := scan_time,
    WATCHDOG := watchdog,
    X := x); // NET_VAR_CONTROL
run := NET_VAR_CONTROL_1.RUN;
error := NET_VAR_CONTROL_1.ERROR;

END_PROGRAM

// POUs/OTHER/NETWORK_VERSION
FUNCTION NETWORK_VERSION : DWORD
VAR_INPUT
	IN : BOOL;
END_VAR

(*
version 1.0	02. feb 2011
programmer 	kst
tested by		oscat

network_version returns the version number in dword format
110 is library version 1.10
if IN = true, the release date will be returned

*)

IF in THEN
	NETWORK_VERSION := DATE_TO_DWORD(D#2016-07-01);
ELSE
	NETWORK_VERSION := 135;
END_IF;

(* revision history
ks	2. feb 2011	rev 1.0
	original version

*)

END_FUNCTION

// POUs/DEMO/RC4_CRYPT_DEMO
PROGRAM RC4_CRYPT_DEMO
VAR
	RC4_CRYPT_STREAM: RC4_CRYPT_STREAM;
	(* buf : ARRAY [0..63] OF BYTE := [107,117,114,116];*) (* kurt *)
	buf : ARRAY [0..63] OF BYTE := [110,60,3,219]; (* crypt *)
	mode: INT;
	key: STRING := '1234';
	size: UDINT := 4;
	pos: UDINT;
END_VAR

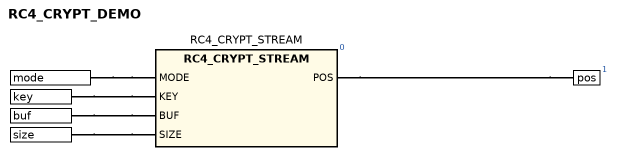
RC4_CRYPT_STREAM(MODE := mode, KEY := key, BUF := buf, SIZE := size);
pos := RC4_CRYPT_STREAM.POS;

END_PROGRAM

// POUs/CONVERT/RC4_CRYPT_STREAM
FUNCTION_BLOCK RC4_CRYPT_STREAM
VAR_IN_OUT
	MODE : INT;
	KEY : STRING(40);
	BUF : ARRAY [0..63] OF BYTE;
	SIZE : UDINT;
END_VAR

VAR_OUTPUT
	POS : UDINT;
END_VAR

VAR
	sbox : ARRAY [0..255] OF BYTE;
	skey : ARRAY [0..255] OF BYTE;
	a : INT;
	b : INT;
	c : INT;
	d : USINT;
	e : USINT;
	end : UDINT;
	v : BYTE;
END_VAR

(*
version 1.0	09. jan. 2010
programmer	ks
tested BY	ks

RC4_CRYPT_STREAM kann einen Datenstrom ver/entschlüsseln mittels der RC4 Stromchiffrierung
*)

CASE MODE OF

